LIN {X 0,Y 347.807,Z 587.248,A -85,B 0,C 180,E1 -13735.5,E2 -13735.5} C_VEL
LIN {X 0,Y 350.643,Z 598.741,A -85,B 0,C 180,E1 -13738.593,E2 -13738.593} C_VEL
LIN {X 0,Y 352.837,Z 609.241,A -85,B 0,C 180,E1 -13741.213,E2 -13741.213} C_VEL
LIN {X 0,Y 353.457,Z 613.128,A -85,B 0,C 180,E1 -13742.144,E2 -13742.144} C_VEL
LIN {X 0,Y 351.63,Z 628.965,A -85,B 0,C 180,E1 -13745.498,E2 -13745.498} C_VEL
LIN {X 0,Y 351.249,Z 632.568,A -85,B 0,C 180,E1 -13746.255,E2 -13746.255} C_VEL
LIN {X 0,Y 354.896,Z 654.897,A -85,B 0,C 180,E1 -13747.117,E2 -13747.117} C_VEL
LIN {X 0,Y 357.589,Z 678.434,A -85,B 0,C 180,E1 -13747.895,E2 -13747.895} C_VEL
LIN {X 0,Y 355.994,Z 743.795,A -85,B 0,C 180,E1 -13749.374,E2 -13749.374} C_VEL
LIN {X 0,Y 355.12,Z 757.95,A -85,B 0,C 180,E1 -13749.926,E2 -13749.926} C_VEL
LIN {X 0,Y 353.991,Z 770.595,A -85,B 0,C 180,E1 -13750.652,E2 -13750.652} C_VEL
LIN {X 0,Y 352.711,Z 782.342,A -85,B 0,C 180,E1 -13751.56,E2 -13751.56} C_VEL
LIN {X 0,Y 351.401,Z 793.761,A -85,B 0,C 180,E1 -13752.693,E2 -13752.693} C_VEL
LIN {X 0,Y 350.119,Z 804.328,A -85,B 0,C 180,E1 -13754.008,E2 -13754.008} C_VEL
LIN {X 0,Y 349.136,Z 813.806,A -85,B 0,C 180,E1 -13755.478,E2 -13755.478} C_VEL
LIN {X 0,Y 348.13,Z 821.311,A -85,B 0,C 180,E1 -13756.873,E2 -13756.873} C_VEL
LIN {X 0,Y 347.268,Z 829.004,A -85,B 0,C 180,E1 -13758.62,E2 -13758.62} C_VEL
LIN {X 0,Y 346.713,Z 836.139,A -85,B 0,C 180,E1 -13760.668,E2 -13760.668} C_VEL
LIN {X 0,Y 346.519,Z 840.885,A -85,B 0,C 180,E1 -13762.425,E2 -13762.425} C_VEL
LIN {X 0,Y 346.403,Z 844.523,A -85,B 0,C 180,E1 -13764.178,E2 -13764.178} C_VEL
LIN {X 0,Y 346.411,Z 846.353,A -85,B 0,C 180,E1 -13765.345,E2 -13765.345} C_VEL
LIN {X 0,Y 346.594,Z 848.779,A -85,B 0,C 180,E1 -13767.676,E2 -13767.676} C_VEL
LIN {X 0,Y 346.623,Z 849.329,A -85,B 0,C 180,E1 -13768.838,E2 -13768.838} C_VEL
LIN {X 0,Y 346.681,Z 849.46,A -85,B 0,C 180,E1 -13770,E2 -13770} C_VEL
LIN {X 0,Y 346.667,Z 849.18,A -85,B 0,C 180,E1 -13771.162,E2 -13771.162} C_VEL
LIN {X 0,Y 346.617,Z 848.487,A -85,B 0,C 180,E1 -13772.324,E2 -13772.324} C_VEL
LIN {X 0,Y 346.504,Z 847.324,A -85,B 0,C 180,E1 -13773.488,E2 -13773.488} C_VEL
LIN {X 0,Y 346.468,Z 844.785,A -85,B 0,C 180,E1 -13775.237,E2 -13775.237} C_VEL
LIN {X 0,Y 346.469,Z 840.184,A -85,B 0,C 180,E1 -13777.576,E2 -13777.576} C_VEL
LIN {X 0,Y 346.71,Z 835.733,A -85,B 0,C 180,E1 -13779.332,E2 -13779.332} C_VEL
LIN {X 0,Y 347.166,Z 830.086,A -85,B 0,C 180,E1 -13781.088,E2 -13781.088} C_VEL
LIN {X 0,Y 348.039,Z 823.071,A -85,B 0,C 180,E1 -13782.834,E2 -13782.834} C_VEL
LIN {X 0,Y 349.063,Z 814.841,A -85,B 0,C 180,E1 -13784.478,E2 -13784.478} C_VEL
LIN {X 0,Y 350.151,Z 805.338,A -85,B 0,C 180,E1 -13786.02,E2 -13786.02} C_VEL
LIN {X 0,Y 351.496,Z 795.505,A -85,B 0,C 180,E1 -13787.302,E2 -13787.302} C_VEL
LIN {X 0,Y 352.903,Z 784.628,A -85,B 0,C 180,E1 -13788.43,E2 -13788.43} C_VEL
LIN {X 0,Y 354.156,Z 772.464,A -85,B 0,C 180,E1 -13789.414,E2 -13789.414} C_VEL
LIN {X 0,Y 355.416,Z 759.627,A -85,B 0,C 180,E1 -13790.17,E2 -13790.17} C_VEL
LIN {X 0,Y 356.266,Z 746.66,A -85,B 0,C 180,E1 -13790.685,E2 -13790.685} C_VEL
LIN {X 0,Y 356.74,Z 726.665,A -85,B 0,C 180,E1 -13791.149,E2 -13791.149} C_VEL
LIN {X 0,Y 357.675,Z 675.14,A -85,B 0,C 180,E1 -13792.209,E2 -13792.209} C_VEL
LIN {X 0,Y 354.114,Z 644.038,A -85,B 0,C 180,E1 -13793.174,E2 -13793.174} C_VEL
LIN {X 0,Y 351.817,Z 628.158,A -85,B 0,C 180,E1 -13793.751,E2 -13793.751} C_VEL
LIN {X 0,Y 353.374,Z 612.718,A -85,B 0,C 180,E1 -13796.495,E2 -13796.495} C_VEL
LIN {X 0,Y 352.12,Z 605.557,A -85,B 0,C 180,E1 -13797.901,E2 -13797.901} C_VEL
LIN {X 0,Y 348.167,Z 588.997,A -85,B 0,C 180,E1 -13801.317,E2 -13801.317} C_VEL
LIN {X 0,Y 347.753,Z 587.169,A -85,B 0,C 180,E1 -13801.753,E2 -13801.753} C_VEL
LIN {X 0,Y 347.788,Z 587.165,A -85,B 0,C 180,E1 -13805.874,E2 -13805.874} C_VEL
LIN {X 0,Y 347.764,Z 587.161,A -85,B 0,C 180,E1 -13808.79,E2 -13808.79} C_VEL
LIN {X 0,Y 347.764,Z 587.16,A -85,B 0,C 180,E1 -13811.827,E2 -13811.827} C_VEL
LIN {X 0,Y 347.796,Z 587.157,A -85,B 0,C 180,E1 -13815.011,E2 -13815.011} C_VEL
LIN {X 0,Y 347.78,Z 587.163,A -85,B 0,C 180,E1 -13818.39,E2 -13818.39} C_VEL
LIN {X 0,Y 347.774,Z 587.162,A -85,B 0,C 180,E1 -13822.009,E2 -13822.009} C_VEL
LIN {X 0,Y 347.739,Z 587.154,A -85,B 0,C 180,E1 -13825.535,E2 -13825.535} C_VEL
LIN {X 0,Y 347.758,Z 587.169,A -85,B 0,C 180,E1 -13828.302,E2 -13828.302} C_VEL
LIN {X 0,Y 347.8,Z 587.145,A -85,B 0,C 180,E1 -13830.989,E2 -13830.989} C_VEL
LIN {X 0,Y 347.825,Z 587.156,A -85,B 0,C 180,E1 -13833.607,E2 -13833.607} C_VEL
LIN {X 0,Y 347.781,Z 587.153,A -85,B 0,C 180,E1 -13836.161,E2 -13836.161} C_VEL
LIN {X 0,Y 347.805,Z 587.158,A -85,B 0,C 180,E1 -13839.909,E2 -13839.909} C_VEL
LIN {X 0,Y 347.858,Z 587.147,A -85,B 0,C 180,E1 -13842.359,E2 -13842.359} C_VEL
LIN {X 0,Y 347.89,Z 587.142,A -85,B 0,C 180,E1 -13845.97,E2 -13845.97} C_VEL
LIN {X 0,Y 347.921,Z 587.137,A -85,B 0,C 180,E1 -13849.525,E2 -13849.525} C_VEL
LIN {X 0,Y 348.086,Z 587.121,A -85,B 0,C 180,E1 -13853.042,E2 -13853.042} C_VEL
LIN {X 0,Y 348.201,Z 587.095,A -85,B 0,C 180,E1 -13857.686,E2 -13857.686} C_VEL
LIN {X 0,Y 348.339,Z 587.084,A -85,B 0,C 180,E1 -13860,E2 -13860} C_VEL
LIN {X 0,Y 348.2,Z 587.111,A -85,B 0,C 180,E1 -13862.314,E2 -13862.314} C_VEL
LIN {X 0,Y 348.085,Z 587.114,A -85,B 0,C 180,E1 -13866.958,E2 -13866.958} C_VEL
LIN {X 0,Y 347.92,Z 587.145,A -85,B 0,C 180,E1 -13870.475,E2 -13870.475} C_VEL
LIN {X 0,Y 347.891,Z 587.142,A -85,B 0,C 180,E1 -13874.15,E2 -13874.15} C_VEL
LIN {X 0,Y 347.884,Z 587.14,A -85,B 0,C 180,E1 -13878.291,E2 -13878.291} C_VEL
LIN {X 0,Y 347.778,Z 587.163,A -85,B 0,C 180,E1 -13881.634,E2 -13881.634} C_VEL
LIN {X 0,Y 347.804,Z 587.15,A -85,B 0,C 180,E1 -13885.109,E2 -13885.109} C_VEL
LIN {X 0,Y 347.806,Z 587.159,A -85,B 0,C 180,E1 -13887.694,E2 -13887.694} C_VEL
LIN {X 0,Y 347.765,Z 587.155,A -85,B 0,C 180,E1 -13890.347,E2 -13890.347} C_VEL
LIN {X 0,Y 347.743,Z 587.159,A -85,B 0,C 180,E1 -13894.045,E2 -13894.045} C_VEL
LIN {X 0,Y 347.758,Z 587.166,A -85,B 0,C 180,E1 -13897.321,E2 -13897.321} C_VEL
LIN {X 0,Y 347.751,Z 587.161,A -85,B 0,C 180,E1 -13900.295,E2 -13900.295} C_VEL
LIN {X 0,Y 347.74,Z 587.15,A -85,B 0,C 180,E1 -13903.406,E2 -13903.406} C_VEL
LIN {X 0,Y 347.725,Z 587.16,A -85,B 0,C 180,E1 -13906.687,E2 -13906.687} C_VEL
LIN {X 0,Y 347.745,Z 587.169,A -85,B 0,C 180,E1 -13910.174,E2 -13910.174} C_VEL
LIN {X 0,Y 347.76,Z 587.156,A -85,B 0,C 180,E1 -13912.68,E2 -13912.68} C_VEL
LIN {X 0,Y 347.77,Z 587.166,A -85,B 0,C 180,E1 -13913.935,E2 -13913.935} C_VEL
LIN {X 0,Y 348.878,Z 590.169,A -85,B 0,C 180,E1 -13914.134,E2 -13914.134} C_VEL
LIN {X 0,Y 356.945,Z 606.471,A -85,B 0,C 180,E1 -13915.183,E2 -13915.183} C_VEL
LIN {X 0,Y 359.514,Z 612.214,A -85,B 0,C 180,E1 -13915.517,E2 -13915.517} C_VEL
LIN {X 0,Y 357.936,Z 684.333,A -85,B 0,C 180,E1 -13916.986,E2 -13916.986} C_VEL
LIN {X 0,Y 357.54,Z 697.812,A -85,B 0,C 180,E1 -13917.464,E2 -13917.464} C_VEL
LIN {X 0,Y 356.928,Z 709.71,A -85,B 0,C 180,E1 -13918.099,E2 -13918.099} C_VEL
LIN {X 0,Y 355.97,Z 721.495,A -85,B 0,C 180,E1 -13918.95,E2 -13918.95} C_VEL
LIN {X 0,Y 354.873,Z 732.621,A -85,B 0,C 180,E1 -13919.997,E2 -13919.997} C_VEL
LIN {X 0,Y 353.582,Z 743.445,A -85,B 0,C 180,E1 -13921.279,E2 -13921.279} C_VEL
LIN {X 0,Y 352.312,Z 752.919,A -85,B 0,C 180,E1 -13922.69,E2 -13922.69} C_VEL
LIN {X 0,Y 351.113,Z 761.41,A -85,B 0,C 180,E1 -13924.255,E2 -13924.255} C_VEL
LIN {X 0,Y 349.923,Z 769.073,A -85,B 0,C 180,E1 -13926.002,E2 -13926.002} C_VEL
LIN {X 0,Y 348.877,Z 775.646,A -85,B 0,C 180,E1 -13927.919,E2 -13927.919} C_VEL
LIN {X 0,Y 348.027,Z 780.921,A -85,B 0,C 180,E1 -13929.923,E2 -13929.923} C_VEL
LIN {X 0,Y 347.426,Z 784.785,A -85,B 0,C 180,E1 -13931.944,E2 -13931.944} C_VEL
LIN {X 0,Y 347.024,Z 786.887,A -85,B 0,C 180,E1 -13933.529,E2 -13933.529} C_VEL
LIN {X 0,Y 346.831,Z 787.974,A -85,B 0,C 180,E1 -13934.727,E2 -13934.727} C_VEL
LIN {X 0,Y 346.636,Z 788.884,A -85,B 0,C 180,E1 -13937.114,E2 -13937.114} C_VEL
LIN {X 0,Y 346.584,Z 788.745,A -85,B 0,C 180,E1 -13938.301,E2 -13938.301} C_VEL
LIN {X 0,Y 346.634,Z 787.198,A -85,B 0,C 180,E1 -13940.666,E2 -13940.666} C_VEL
LIN {X 0,Y 346.765,Z 785.836,A -85,B 0,C 180,E1 -13941.844,E2 -13941.844} C_VEL
LIN {X 0,Y 347.064,Z 782.957,A -85,B 0,C 180,E1 -13943.606,E2 -13943.606} C_VEL
LIN {X 0,Y 347.388,Z 779.064,A -85,B 0,C 180,E1 -13945.358,E2 -13945.358} C_VEL
LIN {X 0,Y 347.813,Z 774.039,A -85,B 0,C 180,E1 -13947.105,E2 -13947.105} C_VEL
LIN {X 0,Y 348.499,Z 767.685,A -85,B 0,C 180,E1 -13948.844,E2 -13948.844} C_VEL
LIN {X 0,Y 349.282,Z 759.809,A -85,B 0,C 180,E1 -13950.576,E2 -13950.576} C_VEL
LIN {X 0,Y 350.172,Z 751.746,A -85,B 0,C 180,E1 -13952.013,E2 -13952.013} C_VEL
LIN {X 0,Y 351.115,Z 741.892,A -85,B 0,C 180,E1 -13953.443,E2 -13953.443} C_VEL
LIN {X 0,Y 352.091,Z 730.83,A -85,B 0,C 180,E1 -13954.723,E2 -13954.723} C_VEL
LIN {X 0,Y 352.973,Z 720.002,A -85,B 0,C 180,E1 -13955.713,E2 -13955.713} C_VEL
LIN {X 0,Y 353.669,Z 707.954,A -85,B 0,C 180,E1 -13956.561,E2 -13956.561} C_VEL
LIN {X 0,Y 354.218,Z 694.721,A -85,B 0,C 180,E1 -13957.231,E2 -13957.231} C_VEL
LIN {X 0,Y 354.53,Z 682.914,A -85,B 0,C 180,E1 -13957.618,E2 -13957.618} C_VEL
LIN {X 0,Y 355.717,Z 608.285,A -85,B 0,C 180,E1 -13959.124,E2 -13959.124} C_VEL
LIN {X 0,Y 350.334,Z 593.661,A -85,B 0,C 180,E1 -13959.725,E2 -13959.725} C_VEL
LIN {X 0,Y 347.964,Z 587.144,A -85,B 0,C 180,E1 -13960.005,E2 -13960.005} C_VEL
LIN {X 0,Y 347.9,Z 587.152,A -85,B 0,C 180,E1 -13964.149,E2 -13964.149} C_VEL
LIN {X 0,Y 347.893,Z 587.152,A -85,B 0,C 180,E1 -13968.29,E2 -13968.29} C_VEL
LIN {X 0,Y 347.867,Z 587.153,A -85,B 0,C 180,E1 -13968.634,E2 -13968.634} C_VEL
LIN {X 0,Y 347.161,Z 587.24,A -85,B 0,C 180,E1 -13969.277,E2 -13969.277} C_VEL
LIN {X 0,Y 344.285,Z 587.601,A -85,B 0,C 180,E1 -13970.284,E2 -13970.284} C_VEL
LIN {X 0,Y 341.403,Z 587.961,A -85,B 0,C 180,E1 -13971.307,E2 -13971.307} C_VEL
LIN {X 0,Y 340.714,Z 588.043,A -85,B 0,C 180,E1 -13971.968,E2 -13971.968} C_VEL
LIN {X 0,Y 340.75,Z 588.037,A -85,B 0,C 180,E1 -13973.203,E2 -13973.203} C_VEL
LIN {X 0,Y 342.594,Z 592.979,A -85,B 0,C 180,E1 -13973.467,E2 -13973.467} C_VEL
LIN {X 0,Y 349.529,Z 610.359,A -85,B 0,C 180,E1 -13974.303,E2 -13974.303} C_VEL
LIN {X 0,Y 348.094,Z 679.063,A -85,B 0,C 180,E1 -13975.827,E2 -13975.827} C_VEL
LIN {X 0,Y 347.807,Z 692.389,A -85,B 0,C 180,E1 -13976.232,E2 -13976.232} C_VEL
LIN {X 0,Y 347.322,Z 705.35,A -85,B 0,C 180,E1 -13976.862,E2 -13976.862} C_VEL
LIN {X 0,Y 346.562,Z 717.77,A -85,B 0,C 180,E1 -13977.698,E2 -13977.698} C_VEL
LIN {X 0,Y 345.658,Z 729.584,A -85,B 0,C 180,E1 -13978.757,E2 -13978.757} C_VEL
LIN {X 0,Y 344.684,Z 740.315,A -85,B 0,C 180,E1 -13979.969,E2 -13979.969} C_VEL
LIN {X 0,Y 343.71,Z 749.983,A -85,B 0,C 180,E1 -13981.319,E2 -13981.319} C_VEL
LIN {X 0,Y 342.79,Z 758.591,A -85,B 0,C 180,E1 -13982.797,E2 -13982.797} C_VEL
LIN {X 0,Y 341.802,Z 767.365,A -85,B 0,C 180,E1 -13984.667,E2 -13984.667} C_VEL
LIN {X 0,Y 341.077,Z 774.28,A -85,B 0,C 180,E1 -13986.524,E2 -13986.524} C_VEL
LIN {X 0,Y 340.513,Z 779.599,A -85,B 0,C 180,E1 -13988.344,E2 -13988.344} C_VEL
LIN {X 0,Y 340.045,Z 783.622,A -85,B 0,C 180,E1 -13990.118,E2 -13990.118} C_VEL
LIN {X 0,Y 339.736,Z 786.566,A -85,B 0,C 180,E1 -13991.865,E2 -13991.865} C_VEL
LIN {X 0,Y 339.522,Z 788.538,A -85,B 0,C 180,E1 -13993.573,E2 -13993.573} C_VEL
LIN {X 0,Y 339.434,Z 789.629,A -85,B 0,C 180,E1 -13995.253,E2 -13995.253} C_VEL
LIN {X 0,Y 339.498,Z 789.921,A -85,B 0,C 180,E1 -13996.911,E2 -13996.911} C_VEL
LIN {X 0,Y 339.603,Z 789.475,A -85,B 0,C 180,E1 -13998.53,E2 -13998.53} C_VEL
LIN {X 0,Y 339.869,Z 788.279,A -85,B 0,C 180,E1 -14000.131,E2 -14000.131} C_VEL
LIN {X 0,Y 340.447,Z 785.112,A -85,B 0,C 180,E1 -14002.484,E2 -14002.484} C_VEL
LIN {X 0,Y 340.931,Z 781.817,A -85,B 0,C 180,E1 -14004.156,E2 -14004.156} C_VEL
LIN {X 0,Y 341.775,Z 776.211,A -85,B 0,C 180,E1 -14006.275,E2 -14006.275} C_VEL
LIN {X 0,Y 342.784,Z 769.782,A -85,B 0,C 180,E1 -14008.133,E2 -14008.133} C_VEL
LIN {X 0,Y 343.98,Z 761.685,A -85,B 0,C 180,E1 -14009.966,E2 -14009.966} C_VEL
LIN {X 0,Y 345.111,Z 753.319,A -85,B 0,C 180,E1 -14011.494,E2 -14011.494} C_VEL
LIN {X 0,Y 346.508,Z 742.896,A -85,B 0,C 180,E1 -14013.019,E2 -14013.019} C_VEL
LIN {X 0,Y 347.632,Z 732.479,A -85,B 0,C 180,E1 -14014.236,E2 -14014.236} C_VEL
LIN {X 0,Y 348.706,Z 721.132,A -85,B 0,C 180,E1 -14015.29,E2 -14015.29} C_VEL
LIN {X 0,Y 349.631,Z 709.216,A -85,B 0,C 180,E1 -14016.138,E2 -14016.138} C_VEL
LIN {X 0,Y 350.174,Z 696.584,A -85,B 0,C 180,E1 -14016.797,E2 -14016.797} C_VEL
LIN {X 0,Y 350.531,Z 684.532,A -85,B 0,C 180,E1 -14017.209,E2 -14017.209} C_VEL
LIN {X 0,Y 352.43,Z 613.13,A -85,B 0,C 180,E1 -14018.855,E2 -14018.855} C_VEL
LIN {X 0,Y 345.875,Z 598.906,A -85,B 0,C 180,E1 -14019.792,E2 -14019.792} C_VEL
LIN {X 0,Y 340.992,Z 589.133,A -85,B 0,C 180,E1 -14020.511,E2 -14020.511} C_VEL
LIN {X 0,Y 340.769,Z 588.039,A -85,B 0,C 180,E1 -14020.576,E2 -14020.576} C_VEL
LIN {X 0,Y 340.779,Z 588.036,A -85,B 0,C 180,E1 -14023.218,E2 -14023.218} C_VEL
LIN {X 0,Y 340.839,Z 588.03,A -85,B 0,C 180,E1 -14026.89,E2 -14026.89} C_VEL
LIN {X 0,Y 340.922,Z 588.017,A -85,B 0,C 180,E1 -14030.508,E2 -14030.508} C_VEL
LIN {X 0,Y 341.07,Z 587.999,A -85,B 0,C 180,E1 -14032.898,E2 -14032.898} C_VEL
LIN {X 0,Y 341.163,Z 587.983,A -85,B 0,C 180,E1 -14037.639,E2 -14037.639} C_VEL
LIN {X 0,Y 341.309,Z 587.969,A -85,B 0,C 180,E1 -14040,E2 -14040} C_VEL
LIN {X 0,Y 341.162,Z 587.99,A -85,B 0,C 180,E1 -14042.361,E2 -14042.361} C_VEL
LIN {X 0,Y 341.057,Z 587.994,A -85,B 0,C 180,E1 -14047.102,E2 -14047.102} C_VEL
LIN {X 0,Y 340.867,Z 588.017,A -85,B 0,C 180,E1 -14050.694,E2 -14050.694} C_VEL
LIN {X 0,Y 340.856,Z 588.016,A -85,B 0,C 180,E1 -14054.325,E2 -14054.325} C_VEL
LIN {X 0,Y 340.831,Z 588.025,A -85,B 0,C 180,E1 -14058.467,E2 -14058.467} C_VEL
LIN {X 0,Y 340.747,Z 588.036,A -85,B 0,C 180,E1 -14061.857,E2 -14061.857} C_VEL
LIN {X 0,Y 340.766,Z 588.036,A -85,B 0,C 180,E1 -14065.665,E2 -14065.665} C_VEL
LIN {X 0,Y 340.736,Z 588.038,A -85,B 0,C 180,E1 -14068.32,E2 -14068.32} C_VEL
LIN {X 0,Y 340.699,Z 588.043,A -85,B 0,C 180,E1 -14071.045,E2 -14071.045} C_VEL
LIN {X 0,Y 340.713,Z 588.044,A -85,B 0,C 180,E1 -14075.28,E2 -14075.28} C_VEL
LIN {X 0,Y 340.714,Z 588.045,A -85,B 0,C 180,E1 -14078.389,E2 -14078.389} C_VEL
LIN {X 0,Y 340.721,Z 588.04,A -85,B 0,C 180,E1 -14081.305,E2 -14081.305} C_VEL
LIN {X 0,Y 340.718,Z 588.045,A -85,B 0,C 180,E1 -14084.533,E2 -14084.533} C_VEL
LIN {X 0,Y 340.731,Z 588.043,A -85,B 0,C 180,E1 -14087.949,E2 -14087.949} C_VEL
LIN {X 0,Y 340.737,Z 588.043,A -85,B 0,C 180,E1 -14091.774,E2 -14091.774} C_VEL
LIN {X 0,Y 340.75,Z 588.112,A -85,B 0,C 180,E1 -14094.905,E2 -14094.905} C_VEL
LIN {X 0,Y 343.72,Z 599.975,A -85,B 0,C 180,E1 -14098.208,E2 -14098.208} C_VEL
LIN {X 0,Y 345.889,Z 610.372,A -85,B 0,C 180,E1 -14100.892,E2 -14100.892} C_VEL
LIN {X 0,Y 346.584,Z 614.357,A -85,B 0,C 180,E1 -14101.872,E2 -14101.872} C_VEL
LIN {X 0,Y 345.433,Z 624.369,A -85,B 0,C 180,E1 -14104.061,E2 -14104.061} C_VEL
LIN {X 0,Y 344.559,Z 631.889,A -85,B 0,C 180,E1 -14105.675,E2 -14105.675} C_VEL
LIN {X 0,Y 348.333,Z 654.595,A -85,B 0,C 180,E1 -14106.582,E2 -14106.582} C_VEL
LIN {X 0,Y 351.166,Z 679.683,A -85,B 0,C 180,E1 -14107.442,E2 -14107.442} C_VEL
LIN {X 0,Y 349.433,Z 743.746,A -85,B 0,C 180,E1 -14108.93,E2 -14108.93} C_VEL
LIN {X 0,Y 348.535,Z 757.689,A -85,B 0,C 180,E1 -14109.491,E2 -14109.491} C_VEL
LIN {X 0,Y 347.438,Z 769.695,A -85,B 0,C 180,E1 -14110.196,E2 -14110.196} C_VEL
LIN {X 0,Y 345.997,Z 782.284,A -85,B 0,C 180,E1 -14111.189,E2 -14111.189} C_VEL
LIN {X 0,Y 344.639,Z 793.599,A -85,B 0,C 180,E1 -14112.342,E2 -14112.342} C_VEL
LIN {X 0,Y 343.274,Z 803.848,A -85,B 0,C 180,E1 -14113.65,E2 -14113.65} C_VEL
LIN {X 0,Y 342.186,Z 813.814,A -85,B 0,C 180,E1 -14115.241,E2 -14115.241} C_VEL
LIN {X 0,Y 341.008,Z 822.306,A -85,B 0,C 180,E1 -14116.897,E2 -14116.897} C_VEL
LIN {X 0,Y 340.158,Z 829.688,A -85,B 0,C 180,E1 -14118.681,E2 -14118.681} C_VEL
LIN {X 0,Y 339.675,Z 835.625,A -85,B 0,C 180,E1 -14120.473,E2 -14120.473} C_VEL
LIN {X 0,Y 339.429,Z 840.345,A -85,B 0,C 180,E1 -14122.266,E2 -14122.266} C_VEL
LIN {X 0,Y 339.327,Z 843.962,A -85,B 0,C 180,E1 -14124.056,E2 -14124.056} C_VEL
LIN {X 0,Y 339.341,Z 845.783,A -85,B 0,C 180,E1 -14125.248,E2 -14125.248} C_VEL
LIN {X 0,Y 339.525,Z 848.183,A -85,B 0,C 180,E1 -14127.627,E2 -14127.627} C_VEL
LIN {X 0,Y 339.551,Z 848.71,A -85,B 0,C 180,E1 -14128.814,E2 -14128.814} C_VEL
LIN {X 0,Y 339.636,Z 848.831,A -85,B 0,C 180,E1 -14130,E2 -14130} C_VEL
LIN {X 0,Y 339.593,Z 848.535,A -85,B 0,C 180,E1 -14131.186,E2 -14131.186} C_VEL
LIN {X 0,Y 339.55,Z 847.823,A -85,B 0,C 180,E1 -14132.372,E2 -14132.372} C_VEL
LIN {X 0,Y 339.416,Z 846.631,A -85,B 0,C 180,E1 -14133.561,E2 -14133.561} C_VEL
LIN {X 0,Y 339.377,Z 842.529,A -85,B 0,C 180,E1 -14136.272,E2 -14136.272} C_VEL
LIN {X 0,Y 339.467,Z 838.381,A -85,B 0,C 180,E1 -14138.333,E2 -14138.333} C_VEL
LIN {X 0,Y 339.8,Z 833.591,A -85,B 0,C 180,E1 -14140.125,E2 -14140.125} C_VEL
LIN {X 0,Y 340.452,Z 827.551,A -85,B 0,C 180,E1 -14141.913,E2 -14141.913} C_VEL
LIN {X 0,Y 341.349,Z 820.058,A -85,B 0,C 180,E1 -14143.696,E2 -14143.696} C_VEL
LIN {X 0,Y 342.453,Z 811.741,A -85,B 0,C 180,E1 -14145.299,E2 -14145.299} C_VEL
LIN {X 0,Y 343.792,Z 802.168,A -85,B 0,C 180,E1 -14146.783,E2 -14146.783} C_VEL
LIN {X 0,Y 345.235,Z 791.706,A -85,B 0,C 180,E1 -14148.086,E2 -14148.086} C_VEL
LIN {X 0,Y 346.7,Z 780.07,A -85,B 0,C 180,E1 -14149.232,E2 -14149.232} C_VEL
LIN {X 0,Y 347.989,Z 768.75,A -85,B 0,C 180,E1 -14150.079,E2 -14150.079} C_VEL
LIN {X 0,Y 349.125,Z 756.052,A -85,B 0,C 180,E1 -14150.78,E2 -14150.78} C_VEL
LIN {X 0,Y 349.929,Z 743.308,A -85,B 0,C 180,E1 -14151.251,E2 -14151.251} C_VEL
LIN {X 0,Y 351.265,Z 675.932,A -85,B 0,C 180,E1 -14152.686,E2 -14152.686} C_VEL
LIN {X 0,Y 348.077,Z 647.6,A -85,B 0,C 180,E1 -14153.584,E2 -14153.584} C_VEL
LIN {X 0,Y 345.076,Z 626.818,A -85,B 0,C 180,E1 -14154.324,E2 -14154.324} C_VEL
LIN {X 0,Y 346.423,Z 613.264,A -85,B 0,C 180,E1 -14156.792,E2 -14156.792} C_VEL
LIN {X 0,Y 343.939,Z 601.661,A -85,B 0,C 180,E1 -14159.156,E2 -14159.156} C_VEL
LIN {X 0,Y 340.702,Z 588.048,A -85,B 0,C 180,E1 -14162.084,E2 -14162.084} C_VEL
LIN {X 0,Y 340.717,Z 588.043,A -85,B 0,C 180,E1 -14165.278,E2 -14165.278} C_VEL
LIN {X 0,Y 340.717,Z 588.038,A -85,B 0,C 180,E1 -14168.387,E2 -14168.387} C_VEL
LIN {X 0,Y 340.73,Z 588.036,A -85,B 0,C 180,E1 -14172.051,E2 -14172.051} C_VEL
LIN {X 0,Y 340.719,Z 588.036,A -85,B 0,C 180,E1 -14175.467,E2 -14175.467} C_VEL
LIN {X 0,Y 340.721,Z 588.04,A -85,B 0,C 180,E1 -14178.695,E2 -14178.695} C_VEL
LIN {X 0,Y 340.736,Z 588.036,A -85,B 0,C 180,E1 -14181.773,E2 -14181.773} C_VEL
LIN {X 0,Y 340.718,Z 588.028,A -85,B 0,C 180,E1 -14185.595,E2 -14185.595} C_VEL
LIN {X 0,Y 340.71,Z 588.041,A -85,B 0,C 180,E1 -14188.956,E2 -14188.956} C_VEL
LIN {X 0,Y 340.773,Z 588.029,A -85,B 0,C 180,E1 -14192.473,E2 -14192.473} C_VEL
LIN {X 0,Y 340.749,Z 588.035,A -85,B 0,C 180,E1 -14195.638,E2 -14195.638} C_VEL
LIN {X 0,Y 340.738,Z 588.037,A -85,B 0,C 180,E1 -14199.474,E2 -14199.474} C_VEL
LIN {X 0,Y 340.85,Z 588.026,A -85,B 0,C 180,E1 -14201.984,E2 -14201.984} C_VEL
LIN {X 0,Y 340.862,Z 588.017,A -85,B 0,C 180,E1 -14205.705,E2 -14205.705} C_VEL
LIN {X 0,Y 340.863,Z 588.017,A -85,B 0,C 180,E1 -14209.306,E2 -14209.306} C_VEL
LIN {X 0,Y 341.054,Z 587.994,A -85,B 0,C 180,E1 -14212.898,E2 -14212.898} C_VEL
LIN {X 0,Y 341.163,Z 587.972,A -85,B 0,C 180,E1 -14217.639,E2 -14217.639} C_VEL
LIN {X 0,Y 341.289,Z 587.962,A -85,B 0,C 180,E1 -14220,E2 -14220} C_VEL
LIN {X 0,Y 341.162,Z 587.989,A -85,B 0,C 180,E1 -14222.361,E2 -14222.361} C_VEL
LIN {X 0,Y 341.053,Z 587.991,A -85,B 0,C 180,E1 -14227.102,E2 -14227.102} C_VEL
LIN {X 0,Y 340.863,Z 588.02,A -85,B 0,C 180,E1 -14230.694,E2 -14230.694} C_VEL
LIN {X 0,Y 340.856,Z 588.019,A -85,B 0,C 180,E1 -14234.325,E2 -14234.325} C_VEL
LIN {X 0,Y 340.83,Z 588.016,A -85,B 0,C 180,E1 -14238.467,E2 -14238.467} C_VEL
LIN {X 0,Y 340.747,Z 588.038,A -85,B 0,C 180,E1 -14241.857,E2 -14241.857} C_VEL
LIN {X 0,Y 340.765,Z 588.031,A -85,B 0,C 180,E1 -14245.665,E2 -14245.665} C_VEL
LIN {X 0,Y 340.736,Z 588.039,A -85,B 0,C 180,E1 -14248.32,E2 -14248.32} C_VEL
LIN {X 0,Y 340.71,Z 588.039,A -85,B 0,C 180,E1 -14251.044,E2 -14251.044} C_VEL
LIN {X 0,Y 340.713,Z 588.039,A -85,B 0,C 180,E1 -14255.28,E2 -14255.28} C_VEL
LIN {X 0,Y 340.713,Z 588.043,A -85,B 0,C 180,E1 -14258.388,E2 -14258.388} C_VEL
LIN {X 0,Y 340.727,Z 588.013,A -85,B 0,C 180,E1 -14262.052,E2 -14262.052} C_VEL
LIN {X 0,Y 340.681,Z 588.049,A -85,B 0,C 180,E1 -14265.462,E2 -14265.462} C_VEL
LIN {X 0,Y 340.683,Z 588.035,A -85,B 0,C 180,E1 -14268.691,E2 -14268.691} C_VEL
LIN {X 0,Y 340.731,Z 588.029,A -85,B 0,C 180,E1 -14271.774,E2 -14271.774} C_VEL
LIN {X 0,Y 340.708,Z 588.042,A -85,B 0,C 180,E1 -14273.339,E2 -14273.339} C_VEL
LIN {X 0,Y 341.743,Z 590.947,A -85,B 0,C 180,E1 -14273.511,E2 -14273.511} C_VEL
LIN {X 0,Y 349.198,Z 605.498,A -85,B 0,C 180,E1 -14274.513,E2 -14274.513} C_VEL
LIN {X 0,Y 353.083,Z 613.998,A -85,B 0,C 180,E1 -14275.033,E2 -14275.033} C_VEL
LIN {X 0,Y 351.511,Z 685.25,A -85,B 0,C 180,E1 -14276.517,E2 -14276.517} C_VEL
LIN {X 0,Y 351.122,Z 698.274,A -85,B 0,C 180,E1 -14276.989,E2 -14276.989} C_VEL
LIN {X 0,Y 350.404,Z 711.311,A -85,B 0,C 180,E1 -14277.706,E2 -14277.706} C_VEL
LIN {X 0,Y 349.335,Z 723.519,A -85,B 0,C 180,E1 -14278.631,E2 -14278.631} C_VEL
LIN {X 0,Y 348.059,Z 735.458,A -85,B 0,C 180,E1 -14279.814,E2 -14279.814} C_VEL
LIN {X 0,Y 346.608,Z 746.437,A -85,B 0,C 180,E1 -14281.213,E2 -14281.213} C_VEL
LIN {X 0,Y 345.285,Z 756.017,A -85,B 0,C 180,E1 -14282.745,E2 -14282.745} C_VEL
LIN {X 0,Y 343.844,Z 765.113,A -85,B 0,C 180,E1 -14284.582,E2 -14284.582} C_VEL
LIN {X 0,Y 342.653,Z 772.362,A -85,B 0,C 180,E1 -14286.425,E2 -14286.425} C_VEL
LIN {X 0,Y 341.704,Z 778.054,A -85,B 0,C 180,E1 -14288.272,E2 -14288.272} C_VEL
LIN {X 0,Y 340.919,Z 782.444,A -85,B 0,C 180,E1 -14290.115,E2 -14290.115} C_VEL
LIN {X 0,Y 340.364,Z 785.694,A -85,B 0,C 180,E1 -14291.958,E2 -14291.958} C_VEL
LIN {X 0,Y 340.044,Z 787.281,A -85,B 0,C 180,E1 -14293.181,E2 -14293.181} C_VEL
LIN {X 0,Y 339.806,Z 788.455,A -85,B 0,C 180,E1 -14294.403,E2 -14294.403} C_VEL
LIN {X 0,Y 339.586,Z 789.445,A -85,B 0,C 180,E1 -14296.583,E2 -14296.583} C_VEL
LIN {X 0,Y 339.522,Z 789.391,A -85,B 0,C 180,E1 -14298.054,E2 -14298.054} C_VEL
LIN {X 0,Y 339.495,Z 788.893,A -85,B 0,C 180,E1 -14299.263,E2 -14299.263} C_VEL
LIN {X 0,Y 339.681,Z 786.656,A -85,B 0,C 180,E1 -14301.673,E2 -14301.673} C_VEL
LIN {X 0,Y 339.865,Z 784.672,A -85,B 0,C 180,E1 -14303.019,E2 -14303.019} C_VEL
LIN {X 0,Y 340.307,Z 780.084,A -85,B 0,C 180,E1 -14305.262,E2 -14305.262} C_VEL
LIN {X 0,Y 340.728,Z 775.188,A -85,B 0,C 180,E1 -14307.044,E2 -14307.044} C_VEL
LIN {X 0,Y 341.42,Z 768.998,A -85,B 0,C 180,E1 -14308.821,E2 -14308.821} C_VEL
LIN {X 0,Y 342.207,Z 761.267,A -85,B 0,C 180,E1 -14310.588,E2 -14310.588} C_VEL
LIN {X 0,Y 343.326,Z 751.629,A -85,B 0,C 180,E1 -14312.346,E2 -14312.346} C_VEL
LIN {X 0,Y 344.274,Z 741.581,A -85,B 0,C 180,E1 -14313.804,E2 -14313.804} C_VEL
LIN {X 0,Y 345.311,Z 730.322,A -85,B 0,C 180,E1 -14315.108,E2 -14315.108} C_VEL
LIN {X 0,Y 346.243,Z 719.127,A -85,B 0,C 180,E1 -14316.117,E2 -14316.117} C_VEL
LIN {X 0,Y 346.945,Z 706.597,A -85,B 0,C 180,E1 -14316.981,E2 -14316.981} C_VEL
LIN {X 0,Y 347.467,Z 694.264,A -85,B 0,C 180,E1 -14317.591,E2 -14317.591} C_VEL
LIN {X 0,Y 347.779,Z 682.133,A -85,B 0,C 180,E1 -14317.972,E2 -14317.972} C_VEL
LIN {X 0,Y 348.895,Z 609.148,A -85,B 0,C 180,E1 -14319.474,E2 -14319.474} C_VEL
LIN {X 0,Y 341,Z 588.596,A -85,B 0,C 180,E1 -14320.367,E2 -14320.367} C_VEL
LIN {X 0,Y 340.901,Z 588.021,A -85,B 0,C 180,E1 -14320.422,E2 -14320.422} C_VEL
LIN {X 0,Y 340.864,Z 588.027,A -85,B 0,C 180,E1 -14324.324,E2 -14324.324} C_VEL
LIN {X 0,Y 340.825,Z 588.03,A -85,B 0,C 180,E1 -14328.618,E2 -14328.618} C_VEL
LIN {X 0,Y 340.714,Z 588.043,A -85,B 0,C 180,E1 -14331.968,E2 -14331.968} C_VEL
LIN {X 0,Y 340.817,Z 588.682,A -85,B 0,C 180,E1 -14332.405,E2 -14332.405} C_VEL
LIN {X 0,Y 341.178,Z 590.863,A -85,B 0,C 180,E1 -14332.893,E2 -14332.893} C_VEL
LIN {X 0,Y 341.778,Z 594.839,A -85,B 0,C 180,E1 -14333.345,E2 -14333.345} C_VEL
LIN {X 0,Y 342.362,Z 599.598,A -85,B 0,C 180,E1 -14333.614,E2 -14333.614} C_VEL
LIN {X 0,Y 343.211,Z 609.814,A -85,B 0,C 180,E1 -14333.908,E2 -14333.908} C_VEL
LIN {X 0,Y 342.867,Z 616.697,A -85,B 0,C 180,E1 -14334.06,E2 -14334.06} C_VEL
LIN {X 0,Y 341.263,Z 685.918,A -85,B 0,C 180,E1 -14335.645,E2 -14335.645} C_VEL
LIN {X 0,Y 340.819,Z 698.833,A -85,B 0,C 180,E1 -14336.152,E2 -14336.152} C_VEL
LIN {X 0,Y 340.225,Z 711.131,A -85,B 0,C 180,E1 -14336.863,E2 -14336.863} C_VEL
LIN {X 0,Y 339.352,Z 723.36,A -85,B 0,C 180,E1 -14337.809,E2 -14337.809} C_VEL
LIN {X 0,Y 338.354,Z 735.477,A -85,B 0,C 180,E1 -14339.046,E2 -14339.046} C_VEL
LIN {X 0,Y 337.327,Z 745.665,A -85,B 0,C 180,E1 -14340.346,E2 -14340.346} C_VEL
LIN {X 0,Y 336.292,Z 755.189,A -85,B 0,C 180,E1 -14341.848,E2 -14341.848} C_VEL
LIN {X 0,Y 335.395,Z 763.086,A -85,B 0,C 180,E1 -14343.378,E2 -14343.378} C_VEL
LIN {X 0,Y 334.571,Z 769.943,A -85,B 0,C 180,E1 -14344.992,E2 -14344.992} C_VEL
LIN {X 0,Y 333.898,Z 776.414,A -85,B 0,C 180,E1 -14346.885,E2 -14346.885} C_VEL
LIN {X 0,Y 333.321,Z 781.375,A -85,B 0,C 180,E1 -14348.727,E2 -14348.727} C_VEL
LIN {X 0,Y 332.845,Z 785.73,A -85,B 0,C 180,E1 -14350.885,E2 -14350.885} C_VEL
LIN {X 0,Y 332.567,Z 788.083,A -85,B 0,C 180,E1 -14352.549,E2 -14352.549} C_VEL
LIN {X 0,Y 332.396,Z 789.662,A -85,B 0,C 180,E1 -14354.244,E2 -14354.244} C_VEL
LIN {X 0,Y 332.386,Z 790.462,A -85,B 0,C 180,E1 -14355.962,E2 -14355.962} C_VEL
LIN {X 0,Y 332.475,Z 790.456,A -85,B 0,C 180,E1 -14357.717,E2 -14357.717} C_VEL
LIN {X 0,Y 332.696,Z 789.584,A -85,B 0,C 180,E1 -14359.505,E2 -14359.505} C_VEL
LIN {X 0,Y 333.082,Z 787.77,A -85,B 0,C 180,E1 -14361.323,E2 -14361.323} C_VEL
LIN {X 0,Y 333.611,Z 784.916,A -85,B 0,C 180,E1 -14363.178,E2 -14363.178} C_VEL
LIN {X 0,Y 334.339,Z 779.998,A -85,B 0,C 180,E1 -14365.42,E2 -14365.42} C_VEL
LIN {X 0,Y 335.322,Z 774.201,A -85,B 0,C 180,E1 -14367.387,E2 -14367.387} C_VEL
LIN {X 0,Y 336.464,Z 767.317,A -85,B 0,C 180,E1 -14369.216,E2 -14369.216} C_VEL
LIN {X 0,Y 337.778,Z 758.515,A -85,B 0,C 180,E1 -14371.063,E2 -14371.063} C_VEL
LIN {X 0,Y 339.022,Z 749.834,A -85,B 0,C 180,E1 -14372.532,E2 -14372.532} C_VEL
LIN {X 0,Y 340.412,Z 739.223,A -85,B 0,C 180,E1 -14373.978,E2 -14373.978} C_VEL
LIN {X 0,Y 341.681,Z 727.549,A -85,B 0,C 180,E1 -14375.229,E2 -14375.229} C_VEL
LIN {X 0,Y 342.732,Z 715.518,A -85,B 0,C 180,E1 -14376.23,E2 -14376.23} C_VEL
LIN {X 0,Y 343.502,Z 702.549,A -85,B 0,C 180,E1 -14377.024,E2 -14377.024} C_VEL
LIN {X 0,Y 343.986,Z 689.266,A -85,B 0,C 180,E1 -14377.583,E2 -14377.583} C_VEL
LIN {X 0,Y 346.117,Z 615.15,A -85,B 0,C 180,E1 -14379.341,E2 -14379.341} C_VEL
LIN {X 0,Y 339.177,Z 600.225,A -85,B 0,C 180,E1 -14380.382,E2 -14380.382} C_VEL
LIN {X 0,Y 334.08,Z 590.245,A -85,B 0,C 180,E1 -14381.161,E2 -14381.161} C_VEL
LIN {X 0,Y 333.767,Z 588.912,A -85,B 0,C 180,E1 -14381.283,E2 -14381.283} C_VEL
LIN {X 0,Y 333.801,Z 588.907,A -85,B 0,C 180,E1 -14385.576,E2 -14385.576} C_VEL
LIN {X 0,Y 333.83,Z 588.903,A -85,B 0,C 180,E1 -14389.078,E2 -14389.078} C_VEL
LIN {X 0,Y 334.019,Z 588.877,A -85,B 0,C 180,E1 -14392.747,E2 -14392.747} C_VEL
LIN {X 0,Y 333.808,Z 588.902,A -85,B 0,C 180,E1 -14395.169,E2 -14395.169} C_VEL
LIN {X 0,Y 334.1,Z 588.863,A -85,B 0,C 180,E1 -14397.589,E2 -14397.589} C_VEL
LIN {X 0,Y 334.259,Z 588.847,A -85,B 0,C 180,E1 -14400,E2 -14400} C_VEL
LIN {X 0,Y 334.1,Z 588.869,A -85,B 0,C 180,E1 -14402.411,E2 -14402.411} C_VEL
LIN {X 0,Y 334.013,Z 588.877,A -85,B 0,C 180,E1 -14406.039,E2 -14406.039} C_VEL
LIN {X 0,Y 333.977,Z 588.883,A -85,B 0,C 180,E1 -14408.501,E2 -14408.501} C_VEL
LIN {X 0,Y 333.788,Z 588.903,A -85,B 0,C 180,E1 -14412.155,E2 -14412.155} C_VEL
LIN {X 0,Y 333.77,Z 588.903,A -85,B 0,C 180,E1 -14415.887,E2 -14415.887} C_VEL
LIN {X 0,Y 333.79,Z 588.904,A -85,B 0,C 180,E1 -14418.656,E2 -14418.656} C_VEL
LIN {X 0,Y 333.686,Z 588.918,A -85,B 0,C 180,E1 -14422.279,E2 -14422.279} C_VEL
LIN {X 0,Y 333.73,Z 588.915,A -85,B 0,C 180,E1 -14426.247,E2 -14426.247} C_VEL
LIN {X 0,Y 333.706,Z 588.918,A -85,B 0,C 180,E1 -14428.973,E2 -14428.973} C_VEL
LIN {X 0,Y 333.641,Z 588.925,A -85,B 0,C 180,E1 -14432.588,E2 -14432.588} C_VEL
LIN {X 0,Y 333.672,Z 588.92,A -85,B 0,C 180,E1 -14436.14,E2 -14436.14} C_VEL
LIN {X 0,Y 333.68,Z 588.916,A -85,B 0,C 180,E1 -14439.188,E2 -14439.188} C_VEL
LIN {X 0,Y 333.685,Z 588.921,A -85,B 0,C 180,E1 -14442.511,E2 -14442.511} C_VEL
LIN {X 0,Y 333.656,Z 588.924,A -85,B 0,C 180,E1 -14445.966,E2 -14445.966} C_VEL
LIN {X 0,Y 333.654,Z 588.923,A -85,B 0,C 180,E1 -14449.314,E2 -14449.314} C_VEL
LIN {X 0,Y 333.654,Z 588.924,A -85,B 0,C 180,E1 -14452.35,E2 -14452.35} C_VEL
LIN {X 0,Y 333.697,Z 589.062,A -85,B 0,C 180,E1 -14454.3,E2 -14454.3} C_VEL
LIN {X 0,Y 336.51,Z 599.941,A -85,B 0,C 180,E1 -14457.468,E2 -14457.468} C_VEL
LIN {X 0,Y 338.982,Z 611.478,A -85,B 0,C 180,E1 -14460.549,E2 -14460.549} C_VEL
LIN {X 0,Y 339.73,Z 617.018,A -85,B 0,C 180,E1 -14461.926,E2 -14461.926} C_VEL
LIN {X 0,Y 337.874,Z 631.12,A -85,B 0,C 180,E1 -14465.048,E2 -14465.048} C_VEL
LIN {X 0,Y 341.799,Z 654.152,A -85,B 0,C 180,E1 -14466.023,E2 -14466.023} C_VEL
LIN {X 0,Y 344.724,Z 679.551,A -85,B 0,C 180,E1 -14466.924,E2 -14466.924} C_VEL
LIN {X 0,Y 342.964,Z 742.944,A -85,B 0,C 180,E1 -14468.434,E2 -14468.434} C_VEL
LIN {X 0,Y 342.019,Z 756.857,A -85,B 0,C 180,E1 -14469.004,E2 -14469.004} C_VEL
LIN {X 0,Y 340.884,Z 768.871,A -85,B 0,C 180,E1 -14469.72,E2 -14469.72} C_VEL
LIN {X 0,Y 339.462,Z 780.661,A -85,B 0,C 180,E1 -14470.656,E2 -14470.656} C_VEL
LIN {X 0,Y 338.031,Z 792.128,A -85,B 0,C 180,E1 -14471.829,E2 -14471.829} C_VEL
LIN {X 0,Y 336.584,Z 802.562,A -85,B 0,C 180,E1 -14473.16,E2 -14473.16} C_VEL
LIN {X 0,Y 335.408,Z 812.318,A -85,B 0,C 180,E1 -14474.72,E2 -14474.72} C_VEL
LIN {X 0,Y 334.184,Z 820.517,A -85,B 0,C 180,E1 -14476.315,E2 -14476.315} C_VEL
LIN {X 0,Y 333.288,Z 828.122,A -85,B 0,C 180,E1 -14478.136,E2 -14478.136} C_VEL
LIN {X 0,Y 332.749,Z 833.303,A -85,B 0,C 180,E1 -14479.658,E2 -14479.658} C_VEL
LIN {X 0,Y 332.416,Z 838.38,A -85,B 0,C 180,E1 -14481.489,E2 -14481.489} C_VEL
LIN {X 0,Y 332.266,Z 842.32,A -85,B 0,C 180,E1 -14483.32,E2 -14483.32} C_VEL
LIN {X 0,Y 332.273,Z 845.215,A -85,B 0,C 180,E1 -14485.147,E2 -14485.147} C_VEL
LIN {X 0,Y 332.269,Z 846.605,A -85,B 0,C 180,E1 -14486.362,E2 -14486.362} C_VEL
LIN {X 0,Y 332.457,Z 847.583,A -85,B 0,C 180,E1 -14487.577,E2 -14487.577} C_VEL
LIN {X 0,Y 332.482,Z 848.092,A -85,B 0,C 180,E1 -14488.789,E2 -14488.789} C_VEL
LIN {X 0,Y 332.574,Z 848.202,A -85,B 0,C 180,E1 -14490,E2 -14490} C_VEL
LIN {X 0,Y 332.521,Z 847.891,A -85,B 0,C 180,E1 -14491.211,E2 -14491.211} C_VEL
LIN {X 0,Y 332.483,Z 847.153,A -85,B 0,C 180,E1 -14492.423,E2 -14492.423} C_VEL
LIN {X 0,Y 332.303,Z 844.329,A -85,B 0,C 180,E1 -14494.853,E2 -14494.853} C_VEL
LIN {X 0,Y 332.27,Z 840.467,A -85,B 0,C 180,E1 -14497.291,E2 -14497.291} C_VEL
LIN {X 0,Y 332.51,Z 836.48,A -85,B 0,C 180,E1 -14499.121,E2 -14499.121} C_VEL
LIN {X 0,Y 333.038,Z 830.365,A -85,B 0,C 180,E1 -14501.256,E2 -14501.256} C_VEL
LIN {X 0,Y 333.953,Z 823.69,A -85,B 0,C 180,E1 -14503.075,E2 -14503.075} C_VEL
LIN {X 0,Y 335.14,Z 815.351,A -85,B 0,C 180,E1 -14504.903,E2 -14504.903} C_VEL
LIN {X 0,Y 336.181,Z 807.004,A -85,B 0,C 180,E1 -14506.392,E2 -14506.392} C_VEL
LIN {X 0,Y 337.77,Z 796.607,A -85,B 0,C 180,E1 -14507.872,E2 -14507.872} C_VEL
LIN {X 0,Y 339.473,Z 784.925,A -85,B 0,C 180,E1 -14509.187,E2 -14509.187} C_VEL
LIN {X 0,Y 340.855,Z 773.221,A -85,B 0,C 180,E1 -14510.203,E2 -14510.203} C_VEL
LIN {X 0,Y 342.189,Z 761.08,A -85,B 0,C 180,E1 -14510.985,E2 -14510.985} C_VEL
LIN {X 0,Y 343.173,Z 748.719,A -85,B 0,C 180,E1 -14511.552,E2 -14511.552} C_VEL
LIN {X 0,Y 343.687,Z 735.08,A -85,B 0,C 180,E1 -14511.938,E2 -14511.938} C_VEL
LIN {X 0,Y 344.863,Z 676.446,A -85,B 0,C 180,E1 -14513.189,E2 -14513.189} C_VEL
LIN {X 0,Y 341.69,Z 648.033,A -85,B 0,C 180,E1 -14514.117,E2 -14514.117} C_VEL
LIN {X 0,Y 338.409,Z 625.201,A -85,B 0,C 180,E1 -14514.969,E2 -14514.969} C_VEL
LIN {X 0,Y 339.49,Z 614.955,A -85,B 0,C 180,E1 -14516.869,E2 -14516.869} C_VEL
LIN {X 0,Y 337.432,Z 604.753,A -85,B 0,C 180,E1 -14518.982,E2 -14518.982} C_VEL
LIN {X 0,Y 333.648,Z 588.926,A -85,B 0,C 180,E1 -14522.442,E2 -14522.442} C_VEL
LIN {X 0,Y 333.676,Z 588.922,A -85,B 0,C 180,E1 -14526.138,E2 -14526.138} C_VEL
LIN {X 0,Y 333.67,Z 588.918,A -85,B 0,C 180,E1 -14529.188,E2 -14529.188} C_VEL
LIN {X 0,Y 333.673,Z 588.917,A -85,B 0,C 180,E1 -14532.507,E2 -14532.507} C_VEL
LIN {X 0,Y 333.666,Z 588.914,A -85,B 0,C 180,E1 -14535.966,E2 -14535.966} C_VEL
LIN {X 0,Y 333.698,Z 588.914,A -85,B 0,C 180,E1 -14539.304,E2 -14539.304} C_VEL
LIN {X 0,Y 333.663,Z 588.92,A -85,B 0,C 180,E1 -14543.166,E2 -14543.166} C_VEL
LIN {X 0,Y 333.636,Z 588.922,A -85,B 0,C 180,E1 -14546.791,E2 -14546.791} C_VEL
LIN {X 0,Y 333.699,Z 588.913,A -85,B 0,C 180,E1 -14549.709,E2 -14549.709} C_VEL
LIN {X 0,Y 333.738,Z 588.904,A -85,B 0,C 180,E1 -14552.401,E2 -14552.401} C_VEL
LIN {X 0,Y 333.72,Z 588.911,A -85,B 0,C 180,E1 -14555.09,E2 -14555.09} C_VEL
LIN {X 0,Y 333.673,Z 588.917,A -85,B 0,C 180,E1 -14559.019,E2 -14559.019} C_VEL
LIN {X 0,Y 333.786,Z 588.904,A -85,B 0,C 180,E1 -14561.589,E2 -14561.589} C_VEL
LIN {X 0,Y 333.801,Z 588.896,A -85,B 0,C 180,E1 -14565.576,E2 -14565.576} C_VEL
LIN {X 0,Y 333.826,Z 588.894,A -85,B 0,C 180,E1 -14569.078,E2 -14569.078} C_VEL
LIN {X 0,Y 334,Z 588.87,A -85,B 0,C 180,E1 -14572.747,E2 -14572.747} C_VEL
LIN {X 0,Y 333.808,Z 588.902,A -85,B 0,C 180,E1 -14575.169,E2 -14575.169} C_VEL
LIN {X 0,Y 334.1,Z 588.851,A -85,B 0,C 180,E1 -14577.589,E2 -14577.589} C_VEL
LIN {X 0,Y 334.24,Z 588.84,A -85,B 0,C 180,E1 -14580,E2 -14580} C_VEL
LIN {X 0,Y 334.124,Z 588.866,A -85,B 0,C 180,E1 -14582.411,E2 -14582.411} C_VEL
LIN {X 0,Y 334.006,Z 588.871,A -85,B 0,C 180,E1 -14587.253,E2 -14587.253} C_VEL
LIN {X 0,Y 333.826,Z 588.893,A -85,B 0,C 180,E1 -14590.922,E2 -14590.922} C_VEL
LIN {X 0,Y 333.801,Z 588.9,A -85,B 0,C 180,E1 -14594.635,E2 -14594.635} C_VEL
LIN {X 0,Y 333.789,Z 588.892,A -85,B 0,C 180,E1 -14598.655,E2 -14598.655} C_VEL
LIN {X 0,Y 333.685,Z 588.919,A -85,B 0,C 180,E1 -14602.279,E2 -14602.279} C_VEL
LIN {X 0,Y 333.729,Z 588.909,A -85,B 0,C 180,E1 -14606.247,E2 -14606.247} C_VEL
LIN {X 0,Y 333.706,Z 588.909,A -85,B 0,C 180,E1 -14608.973,E2 -14608.973} C_VEL
LIN {X 0,Y 333.646,Z 588.925,A -85,B 0,C 180,E1 -14612.59,E2 -14612.59} C_VEL
LIN {X 0,Y 333.671,Z 588.92,A -85,B 0,C 180,E1 -14616.14,E2 -14616.14} C_VEL
LIN {X 0,Y 333.668,Z 588.922,A -85,B 0,C 180,E1 -14619.19,E2 -14619.19} C_VEL
LIN {X 0,Y 333.662,Z 588.893,A -85,B 0,C 180,E1 -14622.507,E2 -14622.507} C_VEL
LIN {X 0,Y 333.619,Z 588.924,A -85,B 0,C 180,E1 -14625.96,E2 -14625.96} C_VEL
LIN {X 0,Y 333.645,Z 588.919,A -85,B 0,C 180,E1 -14629.316,E2 -14629.316} C_VEL
LIN {X 0,Y 333.685,Z 589.032,A -85,B 0,C 180,E1 -14632.7,E2 -14632.7} C_VEL
LIN {X 0,Y 334.721,Z 591.855,A -85,B 0,C 180,E1 -14632.87,E2 -14632.87} C_VEL
LIN {X 0,Y 342.003,Z 605.85,A -85,B 0,C 180,E1 -14633.887,E2 -14633.887} C_VEL
LIN {X 0,Y 346.749,Z 616.062,A -85,B 0,C 180,E1 -14634.544,E2 -14634.544} C_VEL
LIN {X 0,Y 345.155,Z 684.813,A -85,B 0,C 180,E1 -14635.993,E2 -14635.993} C_VEL
LIN {X 0,Y 344.727,Z 698.226,A -85,B 0,C 180,E1 -14636.472,E2 -14636.472} C_VEL
LIN {X 0,Y 344.099,Z 709.845,A -85,B 0,C 180,E1 -14637.099,E2 -14637.099} C_VEL
LIN {X 0,Y 343.039,Z 722.054,A -85,B 0,C 180,E1 -14637.988,E2 -14637.988} C_VEL
LIN {X 0,Y 341.817,Z 733.299,A -85,B 0,C 180,E1 -14639.069,E2 -14639.069} C_VEL
LIN {X 0,Y 340.48,Z 743.539,A -85,B 0,C 180,E1 -14640.305,E2 -14640.305} C_VEL
LIN {X 0,Y 339.264,Z 751.917,A -85,B 0,C 180,E1 -14641.547,E2 -14641.547} C_VEL
LIN {X 0,Y 337.861,Z 761.273,A -85,B 0,C 180,E1 -14643.261,E2 -14643.261} C_VEL
LIN {X 0,Y 336.528,Z 768.823,A -85,B 0,C 180,E1 -14644.983,E2 -14644.983} C_VEL
LIN {X 0,Y 335.25,Z 775.975,A -85,B 0,C 180,E1 -14647.042,E2 -14647.042} C_VEL
LIN {X 0,Y 334.309,Z 781.29,A -85,B 0,C 180,E1 -14649.061,E2 -14649.061} C_VEL
LIN {X 0,Y 333.582,Z 785.125,A -85,B 0,C 180,E1 -14651.004,E2 -14651.004} C_VEL
LIN {X 0,Y 333.083,Z 787.675,A -85,B 0,C 180,E1 -14652.819,E2 -14652.819} C_VEL
LIN {X 0,Y 332.808,Z 788.9,A -85,B 0,C 180,E1 -14654.067,E2 -14654.067} C_VEL
LIN {X 0,Y 332.628,Z 789.704,A -85,B 0,C 180,E1 -14655.313,E2 -14655.313} C_VEL
LIN {X 0,Y 332.529,Z 790.058,A -85,B 0,C 180,E1 -14656.557,E2 -14656.557} C_VEL
LIN {X 0,Y 332.473,Z 790.023,A -85,B 0,C 180,E1 -14657.797,E2 -14657.797} C_VEL
LIN {X 0,Y 332.416,Z 789.606,A -85,B 0,C 180,E1 -14659.031,E2 -14659.031} C_VEL
LIN {X 0,Y 332.479,Z 788.742,A -85,B 0,C 180,E1 -14660.264,E2 -14660.264} C_VEL
LIN {X 0,Y 332.574,Z 787.477,A -85,B 0,C 180,E1 -14661.494,E2 -14661.494} C_VEL
LIN {X 0,Y 332.81,Z 785.392,A -85,B 0,C 180,E1 -14662.983,E2 -14662.983} C_VEL
LIN {X 0,Y 333.226,Z 781.1,A -85,B 0,C 180,E1 -14665.161,E2 -14665.161} C_VEL
LIN {X 0,Y 333.648,Z 776.314,A -85,B 0,C 180,E1 -14666.981,E2 -14666.981} C_VEL
LIN {X 0,Y 334.336,Z 770.268,A -85,B 0,C 180,E1 -14668.796,E2 -14668.796} C_VEL
LIN {X 0,Y 335.141,Z 762.723,A -85,B 0,C 180,E1 -14670.601,E2 -14670.601} C_VEL
LIN {X 0,Y 336.255,Z 753.267,A -85,B 0,C 180,E1 -14672.396,E2 -14672.396} C_VEL
LIN {X 0,Y 337.282,Z 743.504,A -85,B 0,C 180,E1 -14673.883,E2 -14673.883} C_VEL
LIN {X 0,Y 338.28,Z 732.533,A -85,B 0,C 180,E1 -14675.215,E2 -14675.215} C_VEL
LIN {X 0,Y 339.277,Z 721.468,A -85,B 0,C 180,E1 -14676.273,E2 -14676.273} C_VEL
LIN {X 0,Y 340.014,Z 710.006,A -85,B 0,C 180,E1 -14677.124,E2 -14677.124} C_VEL
LIN {X 0,Y 340.57,Z 696.873,A -85,B 0,C 180,E1 -14677.831,E2 -14677.831} C_VEL
LIN {X 0,Y 340.929,Z 684.592,A -85,B 0,C 180,E1 -14678.261,E2 -14678.261} C_VEL
LIN {X 0,Y 342.2,Z 610.829,A -85,B 0,C 180,E1 -14679.81,E2 -14679.81} C_VEL
LIN {X 0,Y 333.963,Z 589.647,A -85,B 0,C 180,E1 -14680.764,E2 -14680.764} C_VEL
LIN {X 0,Y 333.838,Z 588.899,A -85,B 0,C 180,E1 -14680.806,E2 -14680.806} C_VEL
LIN {X 0,Y 333.81,Z 588.904,A -85,B 0,C 180,E1 -14684.634,E2 -14684.634} C_VEL
LIN {X 0,Y 333.798,Z 588.905,A -85,B 0,C 180,E1 -14688.655,E2 -14688.655} C_VEL
LIN {X 0,Y 333.691,Z 588.917,A -85,B 0,C 180,E1 -14692.808,E2 -14692.808} C_VEL
LIN {X 0,Y 336.316,Z 595.799,A -85,B 0,C 180,E1 -14693.151,E2 -14693.151} C_VEL
LIN {X 0,Y 342.912,Z 612.321,A -85,B 0,C 180,E1 -14693.957,E2 -14693.957} C_VEL
LIN {X 0,Y 342.867,Z 616.697,A -85,B 0,C 180,E1 -14694.06,E2 -14694.06} C_VEL
LIN {X 0,Y 342.081,Z 622.525,A -85,B 0,C 180,E1 -14694.156,E2 -14694.156} C_VEL
LIN {X 0,Y 336.205,Z 641.457,A -85,B 0,C 180,E1 -14694.27,E2 -14694.27} C_VEL
LIN {X 0,Y 335.376,Z 647.287,A -85,B 0,C 180,E1 -14694.364,E2 -14694.364} C_VEL
LIN {X 0,Y 334.455,Z 687.48,A -85,B 0,C 180,E1 -14695.327,E2 -14695.327} C_VEL
LIN {X 0,Y 334.023,Z 700.807,A -85,B 0,C 180,E1 -14695.886,E2 -14695.886} C_VEL
LIN {X 0,Y 333.344,Z 712.875,A -85,B 0,C 180,E1 -14696.616,E2 -14696.616} C_VEL
LIN {X 0,Y 332.435,Z 724.814,A -85,B 0,C 180,E1 -14697.585,E2 -14697.585} C_VEL
LIN {X 0,Y 331.413,Z 736.752,A -85,B 0,C 180,E1 -14698.844,E2 -14698.844} C_VEL
LIN {X 0,Y 330.345,Z 747.126,A -85,B 0,C 180,E1 -14700.215,E2 -14700.215} C_VEL
LIN {X 0,Y 329.24,Z 756.747,A -85,B 0,C 180,E1 -14701.802,E2 -14701.802} C_VEL
LIN {X 0,Y 328.183,Z 765.443,A -85,B 0,C 180,E1 -14703.575,E2 -14703.575} C_VEL
LIN {X 0,Y 327.308,Z 772.757,A -85,B 0,C 180,E1 -14705.432,E2 -14705.432} C_VEL
LIN {X 0,Y 326.698,Z 778.457,A -85,B 0,C 180,E1 -14707.254,E2 -14707.254} C_VEL
LIN {X 0,Y 326.146,Z 783.077,A -85,B 0,C 180,E1 -14709.127,E2 -14709.127} C_VEL
LIN {X 0,Y 325.756,Z 786.528,A -85,B 0,C 180,E1 -14710.965,E2 -14710.965} C_VEL
LIN {X 0,Y 325.474,Z 788.96,A -85,B 0,C 180,E1 -14712.763,E2 -14712.763} C_VEL
LIN {X 0,Y 325.316,Z 790.469,A -85,B 0,C 180,E1 -14714.527,E2 -14714.527} C_VEL
LIN {X 0,Y 325.314,Z 791.139,A -85,B 0,C 180,E1 -14716.265,E2 -14716.265} C_VEL
LIN {X 0,Y 325.438,Z 791.039,A -85,B 0,C 180,E1 -14717.974,E2 -14717.974} C_VEL
LIN {X 0,Y 325.653,Z 790.218,A -85,B 0,C 180,E1 -14719.651,E2 -14719.651} C_VEL
LIN {X 0,Y 326.242,Z 787.584,A -85,B 0,C 180,E1 -14722.109,E2 -14722.109} C_VEL
LIN {X 0,Y 326.976,Z 783.345,A -85,B 0,C 180,E1 -14724.526,E2 -14724.526} C_VEL
LIN {X 0,Y 327.921,Z 777.904,A -85,B 0,C 180,E1 -14726.702,E2 -14726.702} C_VEL
LIN {X 0,Y 329.069,Z 771.444,A -85,B 0,C 180,E1 -14728.679,E2 -14728.679} C_VEL
LIN {X 0,Y 330.213,Z 764.612,A -85,B 0,C 180,E1 -14730.342,E2 -14730.342} C_VEL
LIN {X 0,Y 331.549,Z 756.013,A -85,B 0,C 180,E1 -14732.031,E2 -14732.031} C_VEL
LIN {X 0,Y 332.961,Z 746.494,A -85,B 0,C 180,E1 -14733.538,E2 -14733.538} C_VEL
LIN {X 0,Y 334.3,Z 735.865,A -85,B 0,C 180,E1 -14734.896,E2 -14734.896} C_VEL
LIN {X 0,Y 335.509,Z 724.282,A -85,B 0,C 180,E1 -14736.055,E2 -14736.055} C_VEL
LIN {X 0,Y 336.664,Z 711.391,A -85,B 0,C 180,E1 -14737.036,E2 -14737.036} C_VEL
LIN {X 0,Y 337.323,Z 698.36,A -85,B 0,C 180,E1 -14737.752,E2 -14737.752} C_VEL
LIN {X 0,Y 337.747,Z 685.912,A -85,B 0,C 180,E1 -14738.2,E2 -14738.2} C_VEL
LIN {X 0,Y 339.873,Z 617.197,A -85,B 0,C 180,E1 -14739.853,E2 -14739.853} C_VEL
LIN {X 0,Y 332.222,Z 601.041,A -85,B 0,C 180,E1 -14741.042,E2 -14741.042} C_VEL
LIN {X 0,Y 327.917,Z 592.892,A -85,B 0,C 180,E1 -14741.733,E2 -14741.733} C_VEL
LIN {X 0,Y 326.733,Z 589.943,A -85,B 0,C 180,E1 -14741.948,E2 -14741.948} C_VEL
LIN {X 0,Y 326.756,Z 589.785,A -85,B 0,C 180,E1 -14745.433,E2 -14745.433} C_VEL
LIN {X 0,Y 326.766,Z 589.782,A -85,B 0,C 180,E1 -14748.839,E2 -14748.839} C_VEL
LIN {X 0,Y 326.973,Z 589.754,A -85,B 0,C 180,E1 -14752.59,E2 -14752.59} C_VEL
LIN {X 0,Y 326.775,Z 589.778,A -85,B 0,C 180,E1 -14755.065,E2 -14755.065} C_VEL
LIN {X 0,Y 327.041,Z 589.743,A -85,B 0,C 180,E1 -14757.537,E2 -14757.537} C_VEL
LIN {X 0,Y 327.21,Z 589.724,A -85,B 0,C 180,E1 -14760,E2 -14760} C_VEL
LIN {X 0,Y 327.041,Z 589.747,A -85,B 0,C 180,E1 -14762.463,E2 -14762.463} C_VEL
LIN {X 0,Y 326.987,Z 589.75,A -85,B 0,C 180,E1 -14766.169,E2 -14766.169} C_VEL
LIN {X 0,Y 326.907,Z 589.762,A -85,B 0,C 180,E1 -14768.655,E2 -14768.655} C_VEL
LIN {X 0,Y 326.731,Z 589.78,A -85,B 0,C 180,E1 -14772.421,E2 -14772.421} C_VEL
LIN {X 0,Y 326.747,Z 589.779,A -85,B 0,C 180,E1 -14774.958,E2 -14774.958} C_VEL
LIN {X 0,Y 326.727,Z 589.782,A -85,B 0,C 180,E1 -14778.839,E2 -14778.839} C_VEL
LIN {X 0,Y 326.614,Z 589.797,A -85,B 0,C 180,E1 -14782.788,E2 -14782.788} C_VEL
LIN {X 0,Y 326.684,Z 589.791,A -85,B 0,C 180,E1 -14785.484,E2 -14785.484} C_VEL
LIN {X 0,Y 326.655,Z 589.794,A -85,B 0,C 180,E1 -14789.66,E2 -14789.66} C_VEL
LIN {X 0,Y 326.603,Z 589.797,A -85,B 0,C 180,E1 -14794.02,E2 -14794.02} C_VEL
LIN {X 0,Y 326.625,Z 589.799,A -85,B 0,C 180,E1 -14797.24,E2 -14797.24} C_VEL
LIN {X 0,Y 326.631,Z 589.798,A -85,B 0,C 180,E1 -14800.203,E2 -14800.203} C_VEL
LIN {X 0,Y 326.615,Z 589.8,A -85,B 0,C 180,E1 -14803.517,E2 -14803.517} C_VEL
LIN {X 0,Y 326.614,Z 589.803,A -85,B 0,C 180,E1 -14807.021,E2 -14807.021} C_VEL
LIN {X 0,Y 326.641,Z 589.798,A -85,B 0,C 180,E1 -14811.395,E2 -14811.395} C_VEL
LIN {X 0,Y 326.664,Z 589.945,A -85,B 0,C 180,E1 -14813.631,E2 -14813.631} C_VEL
LIN {X 0,Y 329.047,Z 599.073,A -85,B 0,C 180,E1 -14816.407,E2 -14816.407} C_VEL
LIN {X 0,Y 331.508,Z 609.736,A -85,B 0,C 180,E1 -14819.417,E2 -14819.417} C_VEL
LIN {X 0,Y 332.913,Z 618.263,A -85,B 0,C 180,E1 -14821.642,E2 -14821.642} C_VEL
LIN {X 0,Y 331.252,Z 630.368,A -85,B 0,C 180,E1 -14824.388,E2 -14824.388} C_VEL
LIN {X 0,Y 335.59,Z 655.652,A -85,B 0,C 180,E1 -14825.505,E2 -14825.505} C_VEL
LIN {X 0,Y 338.397,Z 681.244,A -85,B 0,C 180,E1 -14826.445,E2 -14826.445} C_VEL
LIN {X 0,Y 336.538,Z 742.237,A -85,B 0,C 180,E1 -14827.921,E2 -14827.921} C_VEL
LIN {X 0,Y 335.565,Z 756.141,A -85,B 0,C 180,E1 -14828.5,E2 -14828.5} C_VEL
LIN {X 0,Y 334.369,Z 768.164,A -85,B 0,C 180,E1 -14829.226,E2 -14829.226} C_VEL
LIN {X 0,Y 332.785,Z 780.755,A -85,B 0,C 180,E1 -14830.252,E2 -14830.252} C_VEL
LIN {X 0,Y 331.303,Z 792.075,A -85,B 0,C 180,E1 -14831.446,E2 -14831.446} C_VEL
LIN {X 0,Y 329.778,Z 802.346,A -85,B 0,C 180,E1 -14832.801,E2 -14832.801} C_VEL
LIN {X 0,Y 328.42,Z 812.762,A -85,B 0,C 180,E1 -14834.532,E2 -14834.532} C_VEL
LIN {X 0,Y 327.055,Z 821.539,A -85,B 0,C 180,E1 -14836.328,E2 -14836.328} C_VEL
LIN {X 0,Y 326.141,Z 828.799,A -85,B 0,C 180,E1 -14838.187,E2 -14838.187} C_VEL
LIN {X 0,Y 325.553,Z 834.657,A -85,B 0,C 180,E1 -14840.055,E2 -14840.055} C_VEL
LIN {X 0,Y 325.277,Z 839.307,A -85,B 0,C 180,E1 -14841.927,E2 -14841.927} C_VEL
LIN {X 0,Y 325.193,Z 842.863,A -85,B 0,C 180,E1 -14843.797,E2 -14843.797} C_VEL
LIN {X 0,Y 325.184,Z 844.656,A -85,B 0,C 180,E1 -14845.041,E2 -14845.041} C_VEL
LIN {X 0,Y 325.185,Z 846.032,A -85,B 0,C 180,E1 -14846.283,E2 -14846.283} C_VEL
LIN {X 0,Y 325.389,Z 846.981,A -85,B 0,C 180,E1 -14847.524,E2 -14847.524} C_VEL
LIN {X 0,Y 325.415,Z 847.476,A -85,B 0,C 180,E1 -14848.763,E2 -14848.763} C_VEL
LIN {X 0,Y 325.514,Z 847.572,A -85,B 0,C 180,E1 -14850,E2 -14850} C_VEL
LIN {X 0,Y 325.451,Z 847.247,A -85,B 0,C 180,E1 -14851.237,E2 -14851.237} C_VEL
LIN {X 0,Y 325.416,Z 846.478,A -85,B 0,C 180,E1 -14852.476,E2 -14852.476} C_VEL
LIN {X 0,Y 325.236,Z 843.676,A -85,B 0,C 180,E1 -14854.958,E2 -14854.958} C_VEL
LIN {X 0,Y 325.17,Z 841.188,A -85,B 0,C 180,E1 -14856.765,E2 -14856.765} C_VEL
LIN {X 0,Y 325.347,Z 837.498,A -85,B 0,C 180,E1 -14858.697,E2 -14858.697} C_VEL
LIN {X 0,Y 325.727,Z 832.806,A -85,B 0,C 180,E1 -14860.568,E2 -14860.568} C_VEL
LIN {X 0,Y 326.646,Z 825.745,A -85,B 0,C 180,E1 -14862.74,E2 -14862.74} C_VEL
LIN {X 0,Y 327.767,Z 818.144,A -85,B 0,C 180,E1 -14864.592,E2 -14864.592} C_VEL
LIN {X 0,Y 328.842,Z 810.395,A -85,B 0,C 180,E1 -14866.131,E2 -14866.131} C_VEL
LIN {X 0,Y 330.335,Z 800.958,A -85,B 0,C 180,E1 -14867.648,E2 -14867.648} C_VEL
LIN {X 0,Y 331.97,Z 790.511,A -85,B 0,C 180,E1 -14868.995,E2 -14868.995} C_VEL
LIN {X 0,Y 333.55,Z 778.901,A -85,B 0,C 180,E1 -14870.183,E2 -14870.183} C_VEL
LIN {X 0,Y 335.098,Z 766.503,A -85,B 0,C 180,E1 -14871.129,E2 -14871.129} C_VEL
LIN {X 0,Y 336.323,Z 753.481,A -85,B 0,C 180,E1 -14871.852,E2 -14871.852} C_VEL
LIN {X 0,Y 337.163,Z 740.879,A -85,B 0,C 180,E1 -14872.302,E2 -14872.302} C_VEL
LIN {X 0,Y 338.56,Z 678.116,A -85,B 0,C 180,E1 -14873.681,E2 -14873.681} C_VEL
LIN {X 0,Y 335.51,Z 649.824,A -85,B 0,C 180,E1 -14874.622,E2 -14874.622} C_VEL
LIN {X 0,Y 331.74,Z 623.694,A -85,B 0,C 180,E1 -14875.615,E2 -14875.615} C_VEL
LIN {X 0,Y 332.511,Z 615.684,A -85,B 0,C 180,E1 -14877.14,E2 -14877.14} C_VEL
LIN {X 0,Y 329.891,Z 603.732,A -85,B 0,C 180,E1 -14879.69,E2 -14879.69} C_VEL
LIN {X 0,Y 326.596,Z 589.803,A -85,B 0,C 180,E1 -14882.83,E2 -14882.83} C_VEL
LIN {X 0,Y 326.612,Z 589.802,A -85,B 0,C 180,E1 -14885.519,E2 -14885.519} C_VEL
LIN {X 0,Y 326.633,Z 589.794,A -85,B 0,C 180,E1 -14889.231,E2 -14889.231} C_VEL
LIN {X 0,Y 326.607,Z 589.8,A -85,B 0,C 180,E1 -14893.517,E2 -14893.517} C_VEL
LIN {X 0,Y 326.624,Z 589.797,A -85,B 0,C 180,E1 -14897.018,E2 -14897.018} C_VEL
LIN {X 0,Y 326.641,Z 589.787,A -85,B 0,C 180,E1 -14900.765,E2 -14900.765} C_VEL
LIN {X 0,Y 326.608,Z 589.789,A -85,B 0,C 180,E1 -14904.48,E2 -14904.48} C_VEL
LIN {X 0,Y 326.61,Z 589.798,A -85,B 0,C 180,E1 -14907.456,E2 -14907.456} C_VEL
LIN {X 0,Y 326.656,Z 589.781,A -85,B 0,C 180,E1 -14910.34,E2 -14910.34} C_VEL
LIN {X 0,Y 326.684,Z 589.792,A -85,B 0,C 180,E1 -14914.516,E2 -14914.516} C_VEL
LIN {X 0,Y 326.639,Z 589.784,A -85,B 0,C 180,E1 -14918.545,E2 -14918.545} C_VEL
LIN {X 0,Y 326.738,Z 589.782,A -85,B 0,C 180,E1 -14921.177,E2 -14921.177} C_VEL
LIN {X 0,Y 326.756,Z 589.773,A -85,B 0,C 180,E1 -14925.433,E2 -14925.433} C_VEL
LIN {X 0,Y 326.762,Z 589.776,A -85,B 0,C 180,E1 -14928.839,E2 -14928.839} C_VEL
LIN {X 0,Y 326.952,Z 589.745,A -85,B 0,C 180,E1 -14932.59,E2 -14932.59} C_VEL
LIN {X 0,Y 326.775,Z 589.779,A -85,B 0,C 180,E1 -14935.065,E2 -14935.065} C_VEL
LIN {X 0,Y 327.041,Z 589.731,A -85,B 0,C 180,E1 -14937.537,E2 -14937.537} C_VEL
LIN {X 0,Y 327.192,Z 589.717,A -85,B 0,C 180,E1 -14940,E2 -14940} C_VEL
LIN {X 0,Y 327.061,Z 589.746,A -85,B 0,C 180,E1 -14942.463,E2 -14942.463} C_VEL
LIN {X 0,Y 326.957,Z 589.74,A -85,B 0,C 180,E1 -14946.615,E2 -14946.615} C_VEL
LIN {X 0,Y 326.907,Z 589.763,A -85,B 0,C 180,E1 -14948.655,E2 -14948.655} C_VEL
LIN {X 0,Y 326.726,Z 589.768,A -85,B 0,C 180,E1 -14952.422,E2 -14952.422} C_VEL
LIN {X 0,Y 326.747,Z 589.782,A -85,B 0,C 180,E1 -14954.958,E2 -14954.958} C_VEL
LIN {X 0,Y 326.726,Z 589.771,A -85,B 0,C 180,E1 -14958.838,E2 -14958.838} C_VEL
LIN {X 0,Y 326.613,Z 589.799,A -85,B 0,C 180,E1 -14962.788,E2 -14962.788} C_VEL
LIN {X 0,Y 326.684,Z 589.782,A -85,B 0,C 180,E1 -14965.484,E2 -14965.484} C_VEL
LIN {X 0,Y 326.656,Z 589.783,A -85,B 0,C 180,E1 -14969.66,E2 -14969.66} C_VEL
LIN {X 0,Y 326.618,Z 589.799,A -85,B 0,C 180,E1 -14972.948,E2 -14972.948} C_VEL
LIN {X 0,Y 326.627,Z 589.799,A -85,B 0,C 180,E1 -14977.047,E2 -14977.047} C_VEL
LIN {X 0,Y 326.6,Z 589.795,A -85,B 0,C 180,E1 -14980.208,E2 -14980.208} C_VEL
LIN {X 0,Y 326.588,Z 589.784,A -85,B 0,C 180,E1 -14983.521,E2 -14983.521} C_VEL
LIN {X 0,Y 326.579,Z 589.788,A -85,B 0,C 180,E1 -14987.028,E2 -14987.028} C_VEL
LIN {X 0,Y 326.609,Z 589.797,A -85,B 0,C 180,E1 -14990.774,E2 -14990.774} C_VEL
LIN {X 0,Y 326.628,Z 589.981,A -85,B 0,C 180,E1 -14992.015,E2 -14992.015} C_VEL
LIN {X 0,Y 327.812,Z 592.961,A -85,B 0,C 180,E1 -14992.211,E2 -14992.211} C_VEL
LIN {X 0,Y 336.24,Z 609.024,A -85,B 0,C 180,E1 -14993.43,E2 -14993.43} C_VEL
LIN {X 0,Y 340.443,Z 618.317,A -85,B 0,C 180,E1 -14994.039,E2 -14994.039} C_VEL
LIN {X 0,Y 338.812,Z 684.628,A -85,B 0,C 180,E1 -14995.457,E2 -14995.457} C_VEL
LIN {X 0,Y 338.409,Z 697.332,A -85,B 0,C 180,E1 -14995.895,E2 -14995.895} C_VEL
LIN {X 0,Y 337.792,Z 708.91,A -85,B 0,C 180,E1 -14996.507,E2 -14996.507} C_VEL
LIN {X 0,Y 336.812,Z 720.406,A -85,B 0,C 180,E1 -14997.323,E2 -14997.323} C_VEL
LIN {X 0,Y 335.54,Z 732.235,A -85,B 0,C 180,E1 -14998.425,E2 -14998.425} C_VEL
LIN {X 0,Y 334.107,Z 742.765,A -85,B 0,C 180,E1 -14999.68,E2 -14999.68} C_VEL
LIN {X 0,Y 332.494,Z 753.327,A -85,B 0,C 180,E1 -15001.258,E2 -15001.258} C_VEL
LIN {X 0,Y 331.232,Z 761.394,A -85,B 0,C 180,E1 -15002.77,E2 -15002.77} C_VEL
LIN {X 0,Y 329.872,Z 768.709,A -85,B 0,C 180,E1 -15004.442,E2 -15004.442} C_VEL
LIN {X 0,Y 328.816,Z 774.427,A -85,B 0,C 180,E1 -15006.041,E2 -15006.041} C_VEL
LIN {X 0,Y 327.744,Z 779.925,A -85,B 0,C 180,E1 -15007.96,E2 -15007.96} C_VEL
LIN {X 0,Y 326.924,Z 784.158,A -85,B 0,C 180,E1 -15009.882,E2 -15009.882} C_VEL
LIN {X 0,Y 326.452,Z 786.588,A -85,B 0,C 180,E1 -15011.308,E2 -15011.308} C_VEL
LIN {X 0,Y 325.816,Z 789.348,A -85,B 0,C 180,E1 -15013.715,E2 -15013.715} C_VEL
LIN {X 0,Y 325.607,Z 790.216,A -85,B 0,C 180,E1 -15014.989,E2 -15014.989} C_VEL
LIN {X 0,Y 325.478,Z 790.653,A -85,B 0,C 180,E1 -15016.332,E2 -15016.332} C_VEL
LIN {X 0,Y 325.341,Z 790.287,A -85,B 0,C 180,E1 -15018.79,E2 -15018.79} C_VEL
LIN {X 0,Y 325.383,Z 789.513,A -85,B 0,C 180,E1 -15020.05,E2 -15020.05} C_VEL
LIN {X 0,Y 325.495,Z 788.293,A -85,B 0,C 180,E1 -15021.307,E2 -15021.307} C_VEL
LIN {X 0,Y 325.74,Z 786.071,A -85,B 0,C 180,E1 -15022.967,E2 -15022.967} C_VEL
LIN {X 0,Y 326.146,Z 782.11,A -85,B 0,C 180,E1 -15025.055,E2 -15025.055} C_VEL
LIN {X 0,Y 326.571,Z 777.43,A -85,B 0,C 180,E1 -15026.916,E2 -15026.916} C_VEL
LIN {X 0,Y 327.254,Z 771.502,A -85,B 0,C 180,E1 -15028.769,E2 -15028.769} C_VEL
LIN {X 0,Y 328.073,Z 764.143,A -85,B 0,C 180,E1 -15030.614,E2 -15030.614} C_VEL
LIN {X 0,Y 329.197,Z 754.866,A -85,B 0,C 180,E1 -15032.447,E2 -15032.447} C_VEL
LIN {X 0,Y 330.245,Z 745.336,A -85,B 0,C 180,E1 -15033.966,E2 -15033.966} C_VEL
LIN {X 0,Y 331.267,Z 734.703,A -85,B 0,C 180,E1 -15035.326,E2 -15035.326} C_VEL
LIN {X 0,Y 332.402,Z 722.65,A -85,B 0,C 180,E1 -15036.526,E2 -15036.526} C_VEL
LIN {X 0,Y 333.18,Z 711.498,A -85,B 0,C 180,E1 -15037.386,E2 -15037.386} C_VEL
LIN {X 0,Y 333.75,Z 698.423,A -85,B 0,C 180,E1 -15038.123,E2 -15038.123} C_VEL
LIN {X 0,Y 334.149,Z 684.966,A -85,B 0,C 180,E1 -15038.613,E2 -15038.613} C_VEL
LIN {X 0,Y 335.393,Z 612.2,A -85,B 0,C 180,E1 -15040.173,E2 -15040.173} C_VEL
LIN {X 0,Y 326.949,Z 590.593,A -85,B 0,C 180,E1 -15041.179,E2 -15041.179} C_VEL
LIN {X 0,Y 326.768,Z 589.78,A -85,B 0,C 180,E1 -15041.239,E2 -15041.239} C_VEL
LIN {X 0,Y 326.756,Z 589.781,A -85,B 0,C 180,E1 -15044.957,E2 -15044.957} C_VEL
LIN {X 0,Y 326.733,Z 589.785,A -85,B 0,C 180,E1 -15048.837,E2 -15048.837} C_VEL
LIN {X 0,Y 326.666,Z 589.879,A -85,B 0,C 180,E1 -15052.372,E2 -15052.372} C_VEL
LIN {X 0,Y 329.25,Z 596.634,A -85,B 0,C 180,E1 -15052.719,E2 -15052.719} C_VEL
LIN {X 0,Y 336.213,Z 614.012,A -85,B 0,C 180,E1 -15053.598,E2 -15053.598} C_VEL
LIN {X 0,Y 335.376,Z 647.287,A -85,B 0,C 180,E1 -15054.364,E2 -15054.364} C_VEL
LIN {X 0,Y 334.549,Z 653.115,A -85,B 0,C 180,E1 -15054.457,E2 -15054.457} C_VEL
LIN {X 0,Y 328.692,Z 672.041,A -85,B 0,C 180,E1 -15054.588,E2 -15054.588} C_VEL
LIN {X 0,Y 327.898,Z 677.867,A -85,B 0,C 180,E1 -15054.688,E2 -15054.688} C_VEL
LIN {X 0,Y 327.577,Z 692.682,A -85,B 0,C 180,E1 -15055.129,E2 -15055.129} C_VEL
LIN {X 0,Y 327.079,Z 704.896,A -85,B 0,C 180,E1 -15055.727,E2 -15055.727} C_VEL
LIN {X 0,Y 326.215,Z 717.857,A -85,B 0,C 180,E1 -15056.614,E2 -15056.614} C_VEL
LIN {X 0,Y 325.224,Z 730.114,A -85,B 0,C 180,E1 -15057.736,E2 -15057.736} C_VEL
LIN {X 0,Y 324.14,Z 741.065,A -85,B 0,C 180,E1 -15059.02,E2 -15059.02} C_VEL
LIN {X 0,Y 322.957,Z 751.696,A -85,B 0,C 180,E1 -15060.575,E2 -15060.575} C_VEL
LIN {X 0,Y 322.054,Z 759.558,A -85,B 0,C 180,E1 -15061.99,E2 -15061.99} C_VEL
LIN {X 0,Y 321.049,Z 767.445,A -85,B 0,C 180,E1 -15063.711,E2 -15063.711} C_VEL
LIN {X 0,Y 320.134,Z 774.69,A -85,B 0,C 180,E1 -15065.681,E2 -15065.681} C_VEL
LIN {X 0,Y 319.505,Z 780.384,A -85,B 0,C 180,E1 -15067.639,E2 -15067.639} C_VEL
LIN {X 0,Y 318.952,Z 785.047,A -85,B 0,C 180,E1 -15069.716,E2 -15069.716} C_VEL
LIN {X 0,Y 318.582,Z 787.903,A -85,B 0,C 180,E1 -15071.437,E2 -15071.437} C_VEL
LIN {X 0,Y 318.335,Z 790.036,A -85,B 0,C 180,E1 -15073.235,E2 -15073.235} C_VEL
LIN {X 0,Y 318.229,Z 791.339,A -85,B 0,C 180,E1 -15075.032,E2 -15075.032} C_VEL
LIN {X 0,Y 318.267,Z 791.838,A -85,B 0,C 180,E1 -15076.8,E2 -15076.8} C_VEL
LIN {X 0,Y 318.453,Z 791.51,A -85,B 0,C 180,E1 -15078.619,E2 -15078.619} C_VEL
LIN {X 0,Y 318.764,Z 790.284,A -85,B 0,C 180,E1 -15080.502,E2 -15080.502} C_VEL
LIN {X 0,Y 319.28,Z 788.102,A -85,B 0,C 180,E1 -15082.412,E2 -15082.412} C_VEL
LIN {X 0,Y 319.882,Z 784.82,A -85,B 0,C 180,E1 -15084.379,E2 -15084.379} C_VEL
LIN {X 0,Y 320.716,Z 780.302,A -85,B 0,C 180,E1 -15086.376,E2 -15086.376} C_VEL
LIN {X 0,Y 321.864,Z 774.294,A -85,B 0,C 180,E1 -15088.396,E2 -15088.396} C_VEL
LIN {X 0,Y 323.239,Z 766.566,A -85,B 0,C 180,E1 -15090.421,E2 -15090.421} C_VEL
LIN {X 0,Y 324.555,Z 758.756,A -85,B 0,C 180,E1 -15092.061,E2 -15092.061} C_VEL
LIN {X 0,Y 325.992,Z 749.733,A -85,B 0,C 180,E1 -15093.599,E2 -15093.599} C_VEL
LIN {X 0,Y 327.49,Z 738.786,A -85,B 0,C 180,E1 -15095.092,E2 -15095.092} C_VEL
LIN {X 0,Y 328.736,Z 728.479,A -85,B 0,C 180,E1 -15096.215,E2 -15096.215} C_VEL
LIN {X 0,Y 329.874,Z 716.884,A -85,B 0,C 180,E1 -15097.211,E2 -15097.211} C_VEL
LIN {X 0,Y 330.728,Z 703.785,A -85,B 0,C 180,E1 -15098.046,E2 -15098.046} C_VEL
LIN {X 0,Y 331.268,Z 690.534,A -85,B 0,C 180,E1 -15098.626,E2 -15098.626} C_VEL
LIN {X 0,Y 333.567,Z 619.08,A -85,B 0,C 180,E1 -15100.402,E2 -15100.402} C_VEL
LIN {X 0,Y 326.035,Z 603.293,A -85,B 0,C 180,E1 -15101.63,E2 -15101.63} C_VEL
LIN {X 0,Y 321.019,Z 594.047,A -85,B 0,C 180,E1 -15102.46,E2 -15102.46} C_VEL
LIN {X 0,Y 319.724,Z 591.179,A -85,B 0,C 180,E1 -15102.696,E2 -15102.696} C_VEL
LIN {X 0,Y 319.64,Z 590.672,A -85,B 0,C 180,E1 -15102.733,E2 -15102.733} C_VEL
LIN {X 0,Y 319.726,Z 590.661,A -85,B 0,C 180,E1 -15106.007,E2 -15106.007} C_VEL
LIN {X 0,Y 319.752,Z 590.655,A -85,B 0,C 180,E1 -15109.873,E2 -15109.873} C_VEL
LIN {X 0,Y 319.927,Z 590.632,A -85,B 0,C 180,E1 -15112.426,E2 -15112.426} C_VEL
LIN {X 0,Y 319.744,Z 590.653,A -85,B 0,C 180,E1 -15114.956,E2 -15114.956} C_VEL
LIN {X 0,Y 319.985,Z 590.622,A -85,B 0,C 180,E1 -15117.482,E2 -15117.482} C_VEL
LIN {X 0,Y 320.161,Z 590.602,A -85,B 0,C 180,E1 -15120,E2 -15120} C_VEL
LIN {X 0,Y 319.985,Z 590.625,A -85,B 0,C 180,E1 -15122.518,E2 -15122.518} C_VEL
LIN {X 0,Y 319.942,Z 590.626,A -85,B 0,C 180,E1 -15126.306,E2 -15126.306} C_VEL
LIN {X 0,Y 319.835,Z 590.641,A -85,B 0,C 180,E1 -15128.848,E2 -15128.848} C_VEL
LIN {X 0,Y 319.678,Z 590.655,A -85,B 0,C 180,E1 -15132.7,E2 -15132.7} C_VEL
LIN {X 0,Y 319.692,Z 590.656,A -85,B 0,C 180,E1 -15135.296,E2 -15135.296} C_VEL
LIN {X 0,Y 319.669,Z 590.659,A -85,B 0,C 180,E1 -15139.255,E2 -15139.255} C_VEL
LIN {X 0,Y 319.564,Z 590.672,A -85,B 0,C 180,E1 -15143.32,E2 -15143.32} C_VEL
LIN {X 0,Y 319.629,Z 590.672,A -85,B 0,C 180,E1 -15146.089,E2 -15146.089} C_VEL
LIN {X 0,Y 319.584,Z 590.677,A -85,B 0,C 180,E1 -15148.934,E2 -15148.934} C_VEL
LIN {X 0,Y 319.528,Z 590.682,A -85,B 0,C 180,E1 -15151.862,E2 -15151.862} C_VEL
LIN {X 0,Y 319.575,Z 590.677,A -85,B 0,C 180,E1 -15155.544,E2 -15155.544} C_VEL
LIN {X 0,Y 319.595,Z 590.676,A -85,B 0,C 180,E1 -15158.005,E2 -15158.005} C_VEL
LIN {X 0,Y 319.592,Z 590.672,A -85,B 0,C 180,E1 -15161.612,E2 -15161.612} C_VEL
LIN {X 0,Y 319.572,Z 590.679,A -85,B 0,C 180,E1 -15165.274,E2 -15165.274} C_VEL
LIN {X 0,Y 319.545,Z 590.685,A -85,B 0,C 180,E1 -15168.716,E2 -15168.716} C_VEL
LIN {X 0,Y 319.58,Z 590.677,A -85,B 0,C 180,E1 -15172.344,E2 -15172.344} C_VEL
LIN {X 0,Y 319.606,Z 590.741,A -85,B 0,C 180,E1 -15172.892,E2 -15172.892} C_VEL
LIN {X 0,Y 322.17,Z 600.511,A -85,B 0,C 180,E1 -15175.992,E2 -15175.992} C_VEL
LIN {X 0,Y 324.585,Z 610.928,A -85,B 0,C 180,E1 -15179.024,E2 -15179.024} C_VEL
LIN {X 0,Y 326.108,Z 619.55,A -85,B 0,C 180,E1 -15181.347,E2 -15181.347} C_VEL
LIN {X 0,Y 324.685,Z 629.612,A -85,B 0,C 180,E1 -15183.698,E2 -15183.698} C_VEL
LIN {X 0,Y 329.092,Z 654.8,A -85,B 0,C 180,E1 -15184.869,E2 -15184.869} C_VEL
LIN {X 0,Y 332.077,Z 681.609,A -85,B 0,C 180,E1 -15185.89,E2 -15185.89} C_VEL
LIN {X 0,Y 330.179,Z 741.239,A -85,B 0,C 180,E1 -15187.375,E2 -15187.375} C_VEL
LIN {X 0,Y 329.108,Z 755.442,A -85,B 0,C 180,E1 -15187.974,E2 -15187.974} C_VEL
LIN {X 0,Y 327.761,Z 768.447,A -85,B 0,C 180,E1 -15188.787,E2 -15188.787} C_VEL
LIN {X 0,Y 326.13,Z 780.851,A -85,B 0,C 180,E1 -15189.831,E2 -15189.831} C_VEL
LIN {X 0,Y 324.588,Z 792.031,A -85,B 0,C 180,E1 -15191.048,E2 -15191.048} C_VEL
LIN {X 0,Y 322.817,Z 803.159,A -85,B 0,C 180,E1 -15192.582,E2 -15192.582} C_VEL
LIN {X 0,Y 321.436,Z 813.266,A -85,B 0,C 180,E1 -15194.334,E2 -15194.334} C_VEL
LIN {X 0,Y 320.116,Z 821.191,A -85,B 0,C 180,E1 -15196.025,E2 -15196.025} C_VEL
LIN {X 0,Y 319.167,Z 828.377,A -85,B 0,C 180,E1 -15197.926,E2 -15197.926} C_VEL
LIN {X 0,Y 318.516,Z 834.182,A -85,B 0,C 180,E1 -15199.833,E2 -15199.833} C_VEL
LIN {X 0,Y 318.21,Z 838.799,A -85,B 0,C 180,E1 -15201.746,E2 -15201.746} C_VEL
LIN {X 0,Y 318.123,Z 842.539,A -85,B 0,C 180,E1 -15203.798,E2 -15203.798} C_VEL
LIN {X 0,Y 318.104,Z 845.462,A -85,B 0,C 180,E1 -15206.2,E2 -15206.2} C_VEL
LIN {X 0,Y 318.303,Z 846.377,A -85,B 0,C 180,E1 -15207.469,E2 -15207.469} C_VEL
LIN {X 0,Y 318.349,Z 846.858,A -85,B 0,C 180,E1 -15208.735,E2 -15208.735} C_VEL
LIN {X 0,Y 318.44,Z 846.938,A -85,B 0,C 180,E1 -15210,E2 -15210} C_VEL
LIN {X 0,Y 318.383,Z 846.594,A -85,B 0,C 180,E1 -15211.265,E2 -15211.265} C_VEL
LIN {X 0,Y 318.35,Z 845.789,A -85,B 0,C 180,E1 -15212.531,E2 -15212.531} C_VEL
LIN {X 0,Y 318.131,Z 841.721,A -85,B 0,C 180,E1 -15216.214,E2 -15216.214} C_VEL
LIN {X 0,Y 318.189,Z 838.329,A -85,B 0,C 180,E1 -15218.254,E2 -15218.254} C_VEL
LIN {X 0,Y 318.52,Z 834.065,A -85,B 0,C 180,E1 -15220.167,E2 -15220.167} C_VEL
LIN {X 0,Y 319.369,Z 827.606,A -85,B 0,C 180,E1 -15222.389,E2 -15222.389} C_VEL
LIN {X 0,Y 320.376,Z 820.595,A -85,B 0,C 180,E1 -15224.287,E2 -15224.287} C_VEL
LIN {X 0,Y 321.652,Z 812.441,A -85,B 0,C 180,E1 -15226.056,E2 -15226.056} C_VEL
LIN {X 0,Y 323.26,Z 802.905,A -85,B 0,C 180,E1 -15227.72,E2 -15227.72} C_VEL
LIN {X 0,Y 324.888,Z 793.098,A -85,B 0,C 180,E1 -15229.097,E2 -15229.097} C_VEL
LIN {X 0,Y 326.504,Z 782.268,A -85,B 0,C 180,E1 -15230.309,E2 -15230.309} C_VEL
LIN {X 0,Y 328.146,Z 770.153,A -85,B 0,C 180,E1 -15231.351,E2 -15231.351} C_VEL
LIN {X 0,Y 329.559,Z 757.433,A -85,B 0,C 180,E1 -15232.159,E2 -15232.159} C_VEL
LIN {X 0,Y 330.55,Z 744.478,A -85,B 0,C 180,E1 -15232.714,E2 -15232.714} C_VEL
LIN {X 0,Y 331.089,Z 726.496,A -85,B 0,C 180,E1 -15233.173,E2 -15233.173} C_VEL
LIN {X 0,Y 332.191,Z 678.121,A -85,B 0,C 180,E1 -15234.241,E2 -15234.241} C_VEL
LIN {X 0,Y 329.176,Z 650.173,A -85,B 0,C 180,E1 -15235.201,E2 -15235.201} C_VEL
LIN {X 0,Y 325.09,Z 622.071,A -85,B 0,C 180,E1 -15236.306,E2 -15236.306} C_VEL
LIN {X 0,Y 325.611,Z 617.555,A -85,B 0,C 180,E1 -15237.181,E2 -15237.181} C_VEL
LIN {X 0,Y 323.27,Z 606.468,A -85,B 0,C 180,E1 -15239.586,E2 -15239.586} C_VEL
LIN {X 0,Y 319.562,Z 590.68,A -85,B 0,C 180,E1 -15243.198,E2 -15243.198} C_VEL
LIN {X 0,Y 319.559,Z 590.681,A -85,B 0,C 180,E1 -15246.426,E2 -15246.426} C_VEL
LIN {X 0,Y 319.562,Z 590.677,A -85,B 0,C 180,E1 -15249.669,E2 -15249.669} C_VEL
LIN {X 0,Y 319.586,Z 590.675,A -85,B 0,C 180,E1 -15253.473,E2 -15253.473} C_VEL
LIN {X 0,Y 319.6,Z 590.672,A -85,B 0,C 180,E1 -15257.024,E2 -15257.024} C_VEL
LIN {X 0,Y 319.581,Z 590.665,A -85,B 0,C 180,E1 -15260.376,E2 -15260.376} C_VEL
LIN {X 0,Y 319.556,Z 590.678,A -85,B 0,C 180,E1 -15263.572,E2 -15263.572} C_VEL
LIN {X 0,Y 319.573,Z 590.671,A -85,B 0,C 180,E1 -15266.685,E2 -15266.685} C_VEL
LIN {X 0,Y 319.588,Z 590.671,A -85,B 0,C 180,E1 -15269.616,E2 -15269.616} C_VEL
LIN {X 0,Y 319.603,Z 590.665,A -85,B 0,C 180,E1 -15272.498,E2 -15272.498} C_VEL
LIN {X 0,Y 319.598,Z 590.67,A -85,B 0,C 180,E1 -15275.303,E2 -15275.303} C_VEL
LIN {X 0,Y 319.59,Z 590.657,A -85,B 0,C 180,E1 -15278.047,E2 -15278.047} C_VEL
LIN {X 0,Y 319.682,Z 590.663,A -85,B 0,C 180,E1 -15280.962,E2 -15280.962} C_VEL
LIN {X 0,Y 319.724,Z 590.647,A -85,B 0,C 180,E1 -15285.276,E2 -15285.276} C_VEL
LIN {X 0,Y 319.745,Z 590.644,A -85,B 0,C 180,E1 -15289.872,E2 -15289.872} C_VEL
LIN {X 0,Y 319.906,Z 590.62,A -85,B 0,C 180,E1 -15292.426,E2 -15292.426} C_VEL
LIN {X 0,Y 319.743,Z 590.656,A -85,B 0,C 180,E1 -15294.956,E2 -15294.956} C_VEL
LIN {X 0,Y 319.985,Z 590.609,A -85,B 0,C 180,E1 -15297.482,E2 -15297.482} C_VEL
LIN {X 0,Y 320.144,Z 590.595,A -85,B 0,C 180,E1 -15300,E2 -15300} C_VEL
LIN {X 0,Y 320.001,Z 590.626,A -85,B 0,C 180,E1 -15302.518,E2 -15302.518} C_VEL
LIN {X 0,Y 319.92,Z 590.615,A -85,B 0,C 180,E1 -15306.605,E2 -15306.605} C_VEL
LIN {X 0,Y 319.835,Z 590.646,A -85,B 0,C 180,E1 -15308.848,E2 -15308.848} C_VEL
LIN {X 0,Y 319.673,Z 590.647,A -85,B 0,C 180,E1 -15312.7,E2 -15312.7} C_VEL
LIN {X 0,Y 319.692,Z 590.664,A -85,B 0,C 180,E1 -15315.296,E2 -15315.296} C_VEL
LIN {X 0,Y 319.667,Z 590.651,A -85,B 0,C 180,E1 -15319.256,E2 -15319.256} C_VEL
LIN {X 0,Y 319.562,Z 590.671,A -85,B 0,C 180,E1 -15323.32,E2 -15323.32} C_VEL
LIN {X 0,Y 319.629,Z 590.666,A -85,B 0,C 180,E1 -15326.089,E2 -15326.089} C_VEL
LIN {X 0,Y 319.584,Z 590.668,A -85,B 0,C 180,E1 -15328.934,E2 -15328.934} C_VEL
LIN {X 0,Y 319.533,Z 590.682,A -85,B 0,C 180,E1 -15331.862,E2 -15331.862} C_VEL
LIN {X 0,Y 319.575,Z 590.674,A -85,B 0,C 180,E1 -15335.544,E2 -15335.544} C_VEL
LIN {X 0,Y 319.578,Z 590.676,A -85,B 0,C 180,E1 -15338.008,E2 -15338.008} C_VEL
LIN {X 0,Y 319.564,Z 590.649,A -85,B 0,C 180,E1 -15341.606,E2 -15341.606} C_VEL
LIN {X 0,Y 319.516,Z 590.687,A -85,B 0,C 180,E1 -15345.264,E2 -15345.264} C_VEL
LIN {X 0,Y 319.525,Z 590.669,A -85,B 0,C 180,E1 -15348.713,E2 -15348.713} C_VEL
LIN {X 0,Y 319.575,Z 590.702,A -85,B 0,C 180,E1 -15351.285,E2 -15351.285} C_VEL
LIN {X 0,Y 320.519,Z 593.464,A -85,B 0,C 180,E1 -15351.459,E2 -15351.459} C_VEL
LIN {X 0,Y 325.286,Z 602.093,A -85,B 0,C 180,E1 -15352.182,E2 -15352.182} C_VEL
LIN {X 0,Y 331.381,Z 614.082,A -85,B 0,C 180,E1 -15353.088,E2 -15353.088} C_VEL
LIN {X 0,Y 334.171,Z 620.396,A -85,B 0,C 180,E1 -15353.508,E2 -15353.508} C_VEL
LIN {X 0,Y 332.495,Z 685.592,A -85,B 0,C 180,E1 -15354.928,E2 -15354.928} C_VEL
LIN {X 0,Y 332.056,Z 698.174,A -85,B 0,C 180,E1 -15355.375,E2 -15355.375} C_VEL
LIN {X 0,Y 331.323,Z 710.618,A -85,B 0,C 180,E1 -15356.055,E2 -15356.055} C_VEL
LIN {X 0,Y 330.205,Z 722.664,A -85,B 0,C 180,E1 -15356.949,E2 -15356.949} C_VEL
LIN {X 0,Y 328.881,Z 734.042,A -85,B 0,C 180,E1 -15358.07,E2 -15358.07} C_VEL
LIN {X 0,Y 327.26,Z 745.341,A -85,B 0,C 180,E1 -15359.484,E2 -15359.484} C_VEL
LIN {X 0,Y 325.753,Z 754.705,A -85,B 0,C 180,E1 -15360.96,E2 -15360.96} C_VEL
LIN {X 0,Y 324.215,Z 763.622,A -85,B 0,C 180,E1 -15362.718,E2 -15362.718} C_VEL
LIN {X 0,Y 322.758,Z 771.054,A -85,B 0,C 180,E1 -15364.53,E2 -15364.53} C_VEL
LIN {X 0,Y 321.641,Z 776.655,A -85,B 0,C 180,E1 -15366.226,E2 -15366.226} C_VEL
LIN {X 0,Y 320.618,Z 781.664,A -85,B 0,C 180,E1 -15368.122,E2 -15368.122} C_VEL
LIN {X 0,Y 319.812,Z 785.62,A -85,B 0,C 180,E1 -15370.086,E2 -15370.086} C_VEL
LIN {X 0,Y 319.171,Z 788.476,A -85,B 0,C 180,E1 -15372.045,E2 -15372.045} C_VEL
LIN {X 0,Y 318.824,Z 789.797,A -85,B 0,C 180,E1 -15373.348,E2 -15373.348} C_VEL
LIN {X 0,Y 318.596,Z 790.712,A -85,B 0,C 180,E1 -15374.651,E2 -15374.651} C_VEL
LIN {X 0,Y 318.416,Z 791.259,A -85,B 0,C 180,E1 -15376.206,E2 -15376.206} C_VEL
LIN {X 0,Y 318.27,Z 790.965,A -85,B 0,C 180,E1 -15378.537,E2 -15378.537} C_VEL
LIN {X 0,Y 318.296,Z 790.251,A -85,B 0,C 180,E1 -15379.826,E2 -15379.826} C_VEL
LIN {X 0,Y 318.404,Z 789.108,A -85,B 0,C 180,E1 -15381.112,E2 -15381.112} C_VEL
LIN {X 0,Y 318.676,Z 786.76,A -85,B 0,C 180,E1 -15382.941,E2 -15382.941} C_VEL
LIN {X 0,Y 319.041,Z 783.12,A -85,B 0,C 180,E1 -15384.945,E2 -15384.945} C_VEL
LIN {X 0,Y 319.499,Z 778.542,A -85,B 0,C 180,E1 -15386.848,E2 -15386.848} C_VEL
LIN {X 0,Y 320.305,Z 771.644,A -85,B 0,C 180,E1 -15389.057,E2 -15389.057} C_VEL
LIN {X 0,Y 321.154,Z 764.155,A -85,B 0,C 180,E1 -15390.94,E2 -15390.94} C_VEL
LIN {X 0,Y 322.354,Z 754.735,A -85,B 0,C 180,E1 -15392.812,E2 -15392.812} C_VEL
LIN {X 0,Y 323.442,Z 745.048,A -85,B 0,C 180,E1 -15394.361,E2 -15394.361} C_VEL
LIN {X 0,Y 324.538,Z 734.143,A -85,B 0,C 180,E1 -15395.748,E2 -15395.748} C_VEL
LIN {X 0,Y 325.613,Z 722.838,A -85,B 0,C 180,E1 -15396.88,E2 -15396.88} C_VEL
LIN {X 0,Y 326.451,Z 710.727,A -85,B 0,C 180,E1 -15397.81,E2 -15397.81} C_VEL
LIN {X 0,Y 327.027,Z 697.651,A -85,B 0,C 180,E1 -15398.535,E2 -15398.535} C_VEL
LIN {X 0,Y 327.415,Z 684.458,A -85,B 0,C 180,E1 -15399,E2 -15399} C_VEL
LIN {X 0,Y 328.791,Z 614.241,A -85,B 0,C 180,E1 -15400.522,E2 -15400.522} C_VEL
LIN {X 0,Y 320.541,Z 593.185,A -85,B 0,C 180,E1 -15401.532,E2 -15401.532} C_VEL
LIN {X 0,Y 319.731,Z 590.658,A -85,B 0,C 180,E1 -15401.651,E2 -15401.651} C_VEL
LIN {X 0,Y 319.701,Z 590.659,A -85,B 0,C 180,E1 -15405.295,E2 -15405.295} C_VEL
LIN {X 0,Y 319.674,Z 590.664,A -85,B 0,C 180,E1 -15409.254,E2 -15409.254} C_VEL
LIN {X 0,Y 319.6,Z 590.675,A -85,B 0,C 180,E1 -15411.909,E2 -15411.909} C_VEL
LIN {X 0,Y 321.687,Z 596.174,A -85,B 0,C 180,E1 -15412.2,E2 -15412.2} C_VEL
LIN {X 0,Y 329.507,Z 615.548,A -85,B 0,C 180,E1 -15413.219,E2 -15413.219} C_VEL
LIN {X 0,Y 327.898,Z 677.867,A -85,B 0,C 180,E1 -15414.688,E2 -15414.688} C_VEL
LIN {X 0,Y 327.061,Z 683.689,A -85,B 0,C 180,E1 -15414.791,E2 -15414.791} C_VEL
LIN {X 0,Y 324.044,Z 693.102,A -85,B 0,C 180,E1 -15414.94,E2 -15414.94} C_VEL
LIN {X 0,Y 321.076,Z 702.431,A -85,B 0,C 180,E1 -15415.229,E2 -15415.229} C_VEL
LIN {X 0,Y 320.224,Z 707.973,A -85,B 0,C 180,E1 -15415.524,E2 -15415.524} C_VEL
LIN {X 0,Y 319.322,Z 719.764,A -85,B 0,C 180,E1 -15416.378,E2 -15416.378} C_VEL
LIN {X 0,Y 318.361,Z 730.906,A -85,B 0,C 180,E1 -15417.44,E2 -15417.44} C_VEL
LIN {X 0,Y 317.148,Z 742.518,A -85,B 0,C 180,E1 -15418.843,E2 -15418.843} C_VEL
LIN {X 0,Y 316.038,Z 752.302,A -85,B 0,C 180,E1 -15420.317,E2 -15420.317} C_VEL
LIN {X 0,Y 314.949,Z 761.356,A -85,B 0,C 180,E1 -15422.009,E2 -15422.009} C_VEL
LIN {X 0,Y 313.783,Z 770.133,A -85,B 0,C 180,E1 -15424.051,E2 -15424.051} C_VEL
LIN {X 0,Y 312.968,Z 776.95,A -85,B 0,C 180,E1 -15426.058,E2 -15426.058} C_VEL
LIN {X 0,Y 312.298,Z 782.223,A -85,B 0,C 180,E1 -15428.034,E2 -15428.034} C_VEL
LIN {X 0,Y 311.811,Z 786.229,A -85,B 0,C 180,E1 -15429.974,E2 -15429.974} C_VEL
LIN {X 0,Y 311.438,Z 789.138,A -85,B 0,C 180,E1 -15431.867,E2 -15431.867} C_VEL
LIN {X 0,Y 311.163,Z 791.599,A -85,B 0,C 180,E1 -15434.44,E2 -15434.44} C_VEL
LIN {X 0,Y 311.156,Z 792.372,A -85,B 0,C 180,E1 -15436.283,E2 -15436.283} C_VEL
LIN {X 0,Y 311.324,Z 792.329,A -85,B 0,C 180,E1 -15438.154,E2 -15438.154} C_VEL
LIN {X 0,Y 311.608,Z 791.42,A -85,B 0,C 180,E1 -15440.069,E2 -15440.069} C_VEL
LIN {X 0,Y 312.268,Z 788.827,A -85,B 0,C 180,E1 -15442.579,E2 -15442.579} C_VEL
LIN {X 0,Y 312.797,Z 786.194,A -85,B 0,C 180,E1 -15444.255,E2 -15444.255} C_VEL
LIN {X 0,Y 313.536,Z 782.537,A -85,B 0,C 180,E1 -15446.031,E2 -15446.031} C_VEL
LIN {X 0,Y 314.632,Z 777.043,A -85,B 0,C 180,E1 -15448.081,E2 -15448.081} C_VEL
LIN {X 0,Y 316.003,Z 769.926,A -85,B 0,C 180,E1 -15450.152,E2 -15450.152} C_VEL
LIN {X 0,Y 317.404,Z 762.233,A -85,B 0,C 180,E1 -15451.933,E2 -15451.933} C_VEL
LIN {X 0,Y 319.033,Z 752.739,A -85,B 0,C 180,E1 -15453.683,E2 -15453.683} C_VEL
LIN {X 0,Y 320.665,Z 742.215,A -85,B 0,C 180,E1 -15455.236,E2 -15455.236} C_VEL
LIN {X 0,Y 321.985,Z 731.893,A -85,B 0,C 180,E1 -15456.45,E2 -15456.45} C_VEL
LIN {X 0,Y 323.229,Z 719.981,A -85,B 0,C 180,E1 -15457.551,E2 -15457.551} C_VEL
LIN {X 0,Y 324.272,Z 707.084,A -85,B 0,C 180,E1 -15458.446,E2 -15458.446} C_VEL
LIN {X 0,Y 324.888,Z 694.196,A -85,B 0,C 180,E1 -15459.068,E2 -15459.068} C_VEL
LIN {X 0,Y 325.501,Z 674.149,A -85,B 0,C 180,E1 -15459.636,E2 -15459.636} C_VEL
LIN {X 0,Y 327.306,Z 620.98,A -85,B 0,C 180,E1 -15460.976,E2 -15460.976} C_VEL
LIN {X 0,Y 319.368,Z 604.545,A -85,B 0,C 180,E1 -15462.329,E2 -15462.329} C_VEL
LIN {X 0,Y 314.065,Z 595.042,A -85,B 0,C 180,E1 -15463.255,E2 -15463.255} C_VEL
LIN {X 0,Y 312.716,Z 592.079,A -85,B 0,C 180,E1 -15463.517,E2 -15463.517} C_VEL
LIN {X 0,Y 312.626,Z 591.544,A -85,B 0,C 180,E1 -15463.596,E2 -15463.596} C_VEL
LIN {X 0,Y 312.63,Z 591.544,A -85,B 0,C 180,E1 -15467.009,E2 -15467.009} C_VEL
LIN {X 0,Y 312.827,Z 591.519,A -85,B 0,C 180,E1 -15471.296,E2 -15471.296} C_VEL
LIN {X 0,Y 312.905,Z 591.509,A -85,B 0,C 180,E1 -15473.552,E2 -15473.552} C_VEL
LIN {X 0,Y 312.932,Z 591.5,A -85,B 0,C 180,E1 -15477.426,E2 -15477.426} C_VEL
LIN {X 0,Y 313.113,Z 591.48,A -85,B 0,C 180,E1 -15480,E2 -15480} C_VEL
LIN {X 0,Y 312.931,Z 591.503,A -85,B 0,C 180,E1 -15482.574,E2 -15482.574} C_VEL
LIN {X 0,Y 312.9,Z 591.502,A -85,B 0,C 180,E1 -15486.448,E2 -15486.448} C_VEL
LIN {X 0,Y 312.781,Z 591.518,A -85,B 0,C 180,E1 -15489.049,E2 -15489.049} C_VEL
LIN {X 0,Y 312.629,Z 591.53,A -85,B 0,C 180,E1 -15492.991,E2 -15492.991} C_VEL
LIN {X 0,Y 312.631,Z 591.535,A -85,B 0,C 180,E1 -15495.65,E2 -15495.65} C_VEL
LIN {X 0,Y 312.625,Z 591.537,A -85,B 0,C 180,E1 -15499.237,E2 -15499.237} C_VEL
LIN {X 0,Y 312.539,Z 591.55,A -85,B 0,C 180,E1 -15502.79,E2 -15502.79} C_VEL
LIN {X 0,Y 312.597,Z 591.547,A -85,B 0,C 180,E1 -15505.936,E2 -15505.936} C_VEL
LIN {X 0,Y 312.54,Z 591.553,A -85,B 0,C 180,E1 -15509.651,E2 -15509.651} C_VEL
LIN {X 0,Y 312.515,Z 591.551,A -85,B 0,C 180,E1 -15513.69,E2 -15513.69} C_VEL
LIN {X 0,Y 312.548,Z 591.552,A -85,B 0,C 180,E1 -15517.382,E2 -15517.382} C_VEL
LIN {X 0,Y 312.522,Z 591.556,A -85,B 0,C 180,E1 -15520.704,E2 -15520.704} C_VEL
LIN {X 0,Y 312.529,Z 591.554,A -85,B 0,C 180,E1 -15524.196,E2 -15524.196} C_VEL
LIN {X 0,Y 312.531,Z 591.556,A -85,B 0,C 180,E1 -15527.909,E2 -15527.909} C_VEL
LIN {X 0,Y 312.577,Z 591.715,A -85,B 0,C 180,E1 -15532.157,E2 -15532.157} C_VEL
LIN {X 0,Y 315.328,Z 602.031,A -85,B 0,C 180,E1 -15535.553,E2 -15535.553} C_VEL
LIN {X 0,Y 317.416,Z 611.009,A -85,B 0,C 180,E1 -15538.275,E2 -15538.275} C_VEL
LIN {X 0,Y 319.027,Z 619.405,A -85,B 0,C 180,E1 -15540.65,E2 -15540.65} C_VEL
LIN {X 0,Y 319.145,Z 622.854,A -85,B 0,C 180,E1 -15541.54,E2 -15541.54} C_VEL
LIN {X 0,Y 318.185,Z 628.933,A -85,B 0,C 180,E1 -15542.974,E2 -15542.974} C_VEL
LIN {X 0,Y 322.558,Z 653.709,A -85,B 0,C 180,E1 -15544.183,E2 -15544.183} C_VEL
LIN {X 0,Y 325.442,Z 678.563,A -85,B 0,C 180,E1 -15545.186,E2 -15545.186} C_VEL
LIN {X 0,Y 325.767,Z 682.849,A -85,B 0,C 180,E1 -15545.338,E2 -15545.338} C_VEL
LIN {X 0,Y 323.865,Z 740.336,A -85,B 0,C 180,E1 -15546.798,E2 -15546.798} C_VEL
LIN {X 0,Y 322.787,Z 754.302,A -85,B 0,C 180,E1 -15547.392,E2 -15547.392} C_VEL
LIN {X 0,Y 321.434,Z 766.925,A -85,B 0,C 180,E1 -15548.18,E2 -15548.18} C_VEL
LIN {X 0,Y 319.7,Z 779.455,A -85,B 0,C 180,E1 -15549.239,E2 -15549.239} C_VEL
LIN {X 0,Y 318.081,Z 790.734,A -85,B 0,C 180,E1 -15550.477,E2 -15550.477} C_VEL
LIN {X 0,Y 316.367,Z 800.981,A -85,B 0,C 180,E1 -15551.881,E2 -15551.881} C_VEL
LIN {X 0,Y 314.996,Z 809.926,A -85,B 0,C 180,E1 -15553.393,E2 -15553.393} C_VEL
LIN {X 0,Y 313.75,Z 818.097,A -85,B 0,C 180,E1 -15555.073,E2 -15555.073} C_VEL
LIN {X 0,Y 312.513,Z 825.771,A -85,B 0,C 180,E1 -15557.004,E2 -15557.004} C_VEL
LIN {X 0,Y 311.658,Z 831.977,A -85,B 0,C 180,E1 -15558.95,E2 -15558.95} C_VEL
LIN {X 0,Y 311.225,Z 836.929,A -85,B 0,C 180,E1 -15560.905,E2 -15560.905} C_VEL
LIN {X 0,Y 311.024,Z 840.756,A -85,B 0,C 180,E1 -15562.861,E2 -15562.861} C_VEL
LIN {X 0,Y 311.022,Z 843.55,A -85,B 0,C 180,E1 -15564.814,E2 -15564.814} C_VEL
LIN {X 0,Y 311.024,Z 844.887,A -85,B 0,C 180,E1 -15566.113,E2 -15566.113} C_VEL
LIN {X 0,Y 311.219,Z 845.775,A -85,B 0,C 180,E1 -15567.411,E2 -15567.411} C_VEL
LIN {X 0,Y 311.285,Z 846.242,A -85,B 0,C 180,E1 -15568.706,E2 -15568.706} C_VEL
LIN {X 0,Y 311.369,Z 846.305,A -85,B 0,C 180,E1 -15570,E2 -15570} C_VEL
LIN {X 0,Y 311.318,Z 845.934,A -85,B 0,C 180,E1 -15571.294,E2 -15571.294} C_VEL
LIN {X 0,Y 311.285,Z 845.1,A -85,B 0,C 180,E1 -15572.588,E2 -15572.588} C_VEL
LIN {X 0,Y 311.047,Z 841.448,A -85,B 0,C 180,E1 -15576.191,E2 -15576.191} C_VEL
LIN {X 0,Y 311.125,Z 837.878,A -85,B 0,C 180,E1 -15578.443,E2 -15578.443} C_VEL
LIN {X 0,Y 311.493,Z 833.664,A -85,B 0,C 180,E1 -15580.399,E2 -15580.399} C_VEL
LIN {X 0,Y 312.402,Z 827.258,A -85,B 0,C 180,E1 -15582.67,E2 -15582.67} C_VEL
LIN {X 0,Y 313.478,Z 820.315,A -85,B 0,C 180,E1 -15584.608,E2 -15584.608} C_VEL
LIN {X 0,Y 314.731,Z 812.593,A -85,B 0,C 180,E1 -15586.349,E2 -15586.349} C_VEL
LIN {X 0,Y 316.475,Z 802.811,A -85,B 0,C 180,E1 -15588.113,E2 -15588.113} C_VEL
LIN {X 0,Y 318.2,Z 793.116,A -85,B 0,C 180,E1 -15589.515,E2 -15589.515} C_VEL
LIN {X 0,Y 319.861,Z 782.504,A -85,B 0,C 180,E1 -15590.75,E2 -15590.75} C_VEL
LIN {X 0,Y 321.554,Z 770.624,A -85,B 0,C 180,E1 -15591.811,E2 -15591.811} C_VEL
LIN {X 0,Y 323.01,Z 758.288,A -85,B 0,C 180,E1 -15592.633,E2 -15592.633} C_VEL
LIN {X 0,Y 324.078,Z 746.061,A -85,B 0,C 180,E1 -15593.204,E2 -15593.204} C_VEL
LIN {X 0,Y 324.639,Z 731.577,A -85,B 0,C 180,E1 -15593.618,E2 -15593.618} C_VEL
LIN {X 0,Y 325.911,Z 678.914,A -85,B 0,C 180,E1 -15594.801,E2 -15594.801} C_VEL
LIN {X 0,Y 322.95,Z 651.067,A -85,B 0,C 180,E1 -15595.783,E2 -15595.783} C_VEL
LIN {X 0,Y 318.494,Z 620.333,A -85,B 0,C 180,E1 -15597.046,E2 -15597.046} C_VEL
LIN {X 0,Y 318.523,Z 617.613,A -85,B 0,C 180,E1 -15597.603,E2 -15597.603} C_VEL
LIN {X 0,Y 315.268,Z 603.192,A -85,B 0,C 180,E1 -15600.844,E2 -15600.844} C_VEL
LIN {X 0,Y 312.539,Z 591.556,A -85,B 0,C 180,E1 -15603.629,E2 -15603.629} C_VEL
LIN {X 0,Y 312.54,Z 591.553,A -85,B 0,C 180,E1 -15607.382,E2 -15607.382} C_VEL
LIN {X 0,Y 312.499,Z 591.556,A -85,B 0,C 180,E1 -15610.706,E2 -15610.706} C_VEL
LIN {X 0,Y 312.527,Z 591.555,A -85,B 0,C 180,E1 -15614.195,E2 -15614.195} C_VEL
LIN {X 0,Y 312.545,Z 591.554,A -85,B 0,C 180,E1 -15617.905,E2 -15617.905} C_VEL
LIN {X 0,Y 312.554,Z 591.548,A -85,B 0,C 180,E1 -15621.904,E2 -15621.904} C_VEL
LIN {X 0,Y 312.502,Z 591.542,A -85,B 0,C 180,E1 -15625.789,E2 -15625.789} C_VEL
LIN {X 0,Y 312.523,Z 591.552,A -85,B 0,C 180,E1 -15628.854,E2 -15628.854} C_VEL
LIN {X 0,Y 312.569,Z 591.534,A -85,B 0,C 180,E1 -15631.824,E2 -15631.824} C_VEL
LIN {X 0,Y 312.579,Z 591.547,A -85,B 0,C 180,E1 -15634.71,E2 -15634.71} C_VEL
LIN {X 0,Y 312.581,Z 591.527,A -85,B 0,C 180,E1 -15637.528,E2 -15637.528} C_VEL
LIN {X 0,Y 312.631,Z 591.539,A -85,B 0,C 180,E1 -15641.656,E2 -15641.656} C_VEL
LIN {X 0,Y 312.687,Z 591.526,A -85,B 0,C 180,E1 -15645.686,E2 -15645.686} C_VEL
LIN {X 0,Y 312.691,Z 591.525,A -85,B 0,C 180,E1 -15649.641,E2 -15649.641} C_VEL
LIN {X 0,Y 312.847,Z 591.498,A -85,B 0,C 180,E1 -15652.254,E2 -15652.254} C_VEL
LIN {X 0,Y 312.713,Z 591.533,A -85,B 0,C 180,E1 -15654.842,E2 -15654.842} C_VEL
LIN {X 0,Y 312.985,Z 591.476,A -85,B 0,C 180,E1 -15658.713,E2 -15658.713} C_VEL
LIN {X 0,Y 312.987,Z 591.497,A -85,B 0,C 180,E1 -15661.287,E2 -15661.287} C_VEL
LIN {X 0,Y 312.69,Z 591.528,A -85,B 0,C 180,E1 -15663.866,E2 -15663.866} C_VEL
LIN {X 0,Y 312.885,Z 591.491,A -85,B 0,C 180,E1 -15666.587,E2 -15666.587} C_VEL
LIN {X 0,Y 312.78,Z 591.525,A -85,B 0,C 180,E1 -15669.049,E2 -15669.049} C_VEL
LIN {X 0,Y 312.626,Z 591.525,A -85,B 0,C 180,E1 -15672.991,E2 -15672.991} C_VEL
LIN {X 0,Y 312.631,Z 591.541,A -85,B 0,C 180,E1 -15675.65,E2 -15675.65} C_VEL
LIN {X 0,Y 312.623,Z 591.528,A -85,B 0,C 180,E1 -15679.236,E2 -15679.236} C_VEL
LIN {X 0,Y 312.539,Z 591.552,A -85,B 0,C 180,E1 -15682.789,E2 -15682.789} C_VEL
LIN {X 0,Y 312.597,Z 591.542,A -85,B 0,C 180,E1 -15685.936,E2 -15685.936} C_VEL
LIN {X 0,Y 312.541,Z 591.54,A -85,B 0,C 180,E1 -15689.65,E2 -15689.65} C_VEL
LIN {X 0,Y 312.515,Z 591.548,A -85,B 0,C 180,E1 -15693.69,E2 -15693.69} C_VEL
LIN {X 0,Y 312.536,Z 591.553,A -85,B 0,C 180,E1 -15697.384,E2 -15697.384} C_VEL
LIN {X 0,Y 312.496,Z 591.539,A -85,B 0,C 180,E1 -15700.708,E2 -15700.708} C_VEL
LIN {X 0,Y 312.51,Z 591.549,A -85,B 0,C 180,E1 -15704.199,E2 -15704.199} C_VEL
LIN {X 0,Y 312.483,Z 591.54,A -85,B 0,C 180,E1 -15707.919,E2 -15707.919} C_VEL
LIN {X 0,Y 312.525,Z 591.701,A -85,B 0,C 180,E1 -15710.524,E2 -15710.524} C_VEL
LIN {X 0,Y 313.692,Z 594.676,A -85,B 0,C 180,E1 -15710.736,E2 -15710.736} C_VEL
LIN {X 0,Y 318.223,Z 602.7,A -85,B 0,C 180,E1 -15711.45,E2 -15711.45} C_VEL
LIN {X 0,Y 325.752,Z 617.456,A -85,B 0,C 180,E1 -15712.615,E2 -15712.615} C_VEL
LIN {X 0,Y 327.9,Z 622.043,A -85,B 0,C 180,E1 -15712.945,E2 -15712.945} C_VEL
LIN {X 0,Y 326.22,Z 685.046,A -85,B 0,C 180,E1 -15714.34,E2 -15714.34} C_VEL
LIN {X 0,Y 325.751,Z 698.274,A -85,B 0,C 180,E1 -15714.797,E2 -15714.797} C_VEL
LIN {X 0,Y 324.995,Z 710.958,A -85,B 0,C 180,E1 -15715.498,E2 -15715.498} C_VEL
LIN {X 0,Y 323.834,Z 722.981,A -85,B 0,C 180,E1 -15716.399,E2 -15716.399} C_VEL
LIN {X 0,Y 322.455,Z 734.437,A -85,B 0,C 180,E1 -15717.541,E2 -15717.541} C_VEL
LIN {X 0,Y 320.802,Z 745.552,A -85,B 0,C 180,E1 -15718.95,E2 -15718.95} C_VEL
LIN {X 0,Y 319.319,Z 754.241,A -85,B 0,C 180,E1 -15720.317,E2 -15720.317} C_VEL
LIN {X 0,Y 317.791,Z 762.915,A -85,B 0,C 180,E1 -15722.006,E2 -15722.006} C_VEL
LIN {X 0,Y 316.13,Z 770.959,A -85,B 0,C 180,E1 -15723.956,E2 -15723.956} C_VEL
LIN {X 0,Y 314.981,Z 776.486,A -85,B 0,C 180,E1 -15725.621,E2 -15725.621} C_VEL
LIN {X 0,Y 313.813,Z 781.812,A -85,B 0,C 180,E1 -15727.622,E2 -15727.622} C_VEL
LIN {X 0,Y 312.95,Z 785.884,A -85,B 0,C 180,E1 -15729.63,E2 -15729.63} C_VEL
LIN {X 0,Y 312.241,Z 788.844,A -85,B 0,C 180,E1 -15731.633,E2 -15731.633} C_VEL
LIN {X 0,Y 311.845,Z 790.248,A -85,B 0,C 180,E1 -15732.964,E2 -15732.964} C_VEL
LIN {X 0,Y 311.418,Z 791.772,A -85,B 0,C 180,E1 -15735.627,E2 -15735.627} C_VEL
LIN {X 0,Y 311.283,Z 791.926,A -85,B 0,C 180,E1 -15736.952,E2 -15736.952} C_VEL
LIN {X 0,Y 311.225,Z 790.973,A -85,B 0,C 180,E1 -15739.592,E2 -15739.592} C_VEL
LIN {X 0,Y 311.307,Z 789.914,A -85,B 0,C 180,E1 -15740.908,E2 -15740.908} C_VEL
LIN {X 0,Y 311.606,Z 787.43,A -85,B 0,C 180,E1 -15742.925,E2 -15742.925} C_VEL
LIN {X 0,Y 311.922,Z 784.117,A -85,B 0,C 180,E1 -15744.829,E2 -15744.829} C_VEL
LIN {X 0,Y 312.429,Z 779.65,A -85,B 0,C 180,E1 -15746.776,E2 -15746.776} C_VEL
LIN {X 0,Y 313.227,Z 772.873,A -85,B 0,C 180,E1 -15749.036,E2 -15749.036} C_VEL
LIN {X 0,Y 314.088,Z 765.55,A -85,B 0,C 180,E1 -15750.962,E2 -15750.962} C_VEL
LIN {X 0,Y 315.102,Z 758.037,A -85,B 0,C 180,E1 -15752.557,E2 -15752.557} C_VEL
LIN {X 0,Y 316.289,Z 747.875,A -85,B 0,C 180,E1 -15754.301,E2 -15754.301} C_VEL
LIN {X 0,Y 317.385,Z 737.593,A -85,B 0,C 180,E1 -15755.719,E2 -15755.719} C_VEL
LIN {X 0,Y 318.442,Z 727.196,A -85,B 0,C 180,E1 -15756.86,E2 -15756.86} C_VEL
LIN {X 0,Y 319.438,Z 714.901,A -85,B 0,C 180,E1 -15757.903,E2 -15757.903} C_VEL
LIN {X 0,Y 320.102,Z 701.944,A -85,B 0,C 180,E1 -15758.721,E2 -15758.721} C_VEL
LIN {X 0,Y 320.564,Z 688.69,A -85,B 0,C 180,E1 -15759.265,E2 -15759.265} C_VEL
LIN {X 0,Y 321.972,Z 615.324,A -85,B 0,C 180,E1 -15760.92,E2 -15760.92} C_VEL
LIN {X 0,Y 313.349,Z 593.768,A -85,B 0,C 180,E1 -15762,E2 -15762} C_VEL
LIN {X 0,Y 312.695,Z 591.537,A -85,B 0,C 180,E1 -15762.102,E2 -15762.102} C_VEL
LIN {X 0,Y 312.64,Z 591.538,A -85,B 0,C 180,E1 -15765.649,E2 -15765.649} C_VEL
LIN {X 0,Y 312.653,Z 591.539,A -85,B 0,C 180,E1 -15769.248,E2 -15769.248} C_VEL
LIN {X 0,Y 312.553,Z 591.549,A -85,B 0,C 180,E1 -15771.431,E2 -15771.431} C_VEL
LIN {X 0,Y 314.373,Z 596.455,A -85,B 0,C 180,E1 -15771.71,E2 -15771.71} C_VEL
LIN {X 0,Y 322.779,Z 617.106,A -85,B 0,C 180,E1 -15772.821,E2 -15772.821} C_VEL
LIN {X 0,Y 320.965,Z 688.529,A -85,B 0,C 180,E1 -15774.584,E2 -15774.584} C_VEL
LIN {X 0,Y 320.506,Z 702.131,A -85,B 0,C 180,E1 -15775.181,E2 -15775.181} C_VEL
LIN {X 0,Y 320.224,Z 707.973,A -85,B 0,C 180,E1 -15775.524,E2 -15775.524} C_VEL
LIN {X 0,Y 319.228,Z 713.521,A -85,B 0,C 180,E1 -15775.851,E2 -15775.851} C_VEL
LIN {X 0,Y 315.727,Z 722.355,A -85,B 0,C 180,E1 -15776.384,E2 -15776.384} C_VEL
LIN {X 0,Y 312.171,Z 730.826,A -85,B 0,C 180,E1 -15777.061,E2 -15777.061} C_VEL
LIN {X 0,Y 311.098,Z 735.797,A -85,B 0,C 180,E1 -15777.609,E2 -15777.609} C_VEL
LIN {X 0,Y 309.951,Z 746.148,A -85,B 0,C 180,E1 -15778.99,E2 -15778.99} C_VEL
LIN {X 0,Y 308.696,Z 756.341,A -85,B 0,C 180,E1 -15780.675,E2 -15780.675} C_VEL
LIN {X 0,Y 307.674,Z 764.376,A -85,B 0,C 180,E1 -15782.31,E2 -15782.31} C_VEL
LIN {X 0,Y 306.517,Z 772.525,A -85,B 0,C 180,E1 -15784.368,E2 -15784.368} C_VEL
LIN {X 0,Y 305.76,Z 779.007,A -85,B 0,C 180,E1 -15786.439,E2 -15786.439} C_VEL
LIN {X 0,Y 305.129,Z 783.968,A -85,B 0,C 180,E1 -15788.453,E2 -15788.453} C_VEL
LIN {X 0,Y 304.629,Z 787.674,A -85,B 0,C 180,E1 -15790.418,E2 -15790.418} C_VEL
LIN {X 0,Y 304.282,Z 790.324,A -85,B 0,C 180,E1 -15792.345,E2 -15792.345} C_VEL
LIN {X 0,Y 304.095,Z 792.054,A -85,B 0,C 180,E1 -15794.238,E2 -15794.238} C_VEL
LIN {X 0,Y 304.077,Z 792.951,A -85,B 0,C 180,E1 -15796.102,E2 -15796.102} C_VEL
LIN {X 0,Y 304.227,Z 793.059,A -85,B 0,C 180,E1 -15797.938,E2 -15797.938} C_VEL
LIN {X 0,Y 304.504,Z 792.372,A -85,B 0,C 180,E1 -15799.741,E2 -15799.741} C_VEL
LIN {X 0,Y 305.165,Z 789.965,A -85,B 0,C 180,E1 -15802.429,E2 -15802.429} C_VEL
LIN {X 0,Y 306.025,Z 786.068,A -85,B 0,C 180,E1 -15804.961,E2 -15804.961} C_VEL
LIN {X 0,Y 307.097,Z 780.967,A -85,B 0,C 180,E1 -15807.272,E2 -15807.272} C_VEL
LIN {X 0,Y 308.526,Z 774.224,A -85,B 0,C 180,E1 -15809.547,E2 -15809.547} C_VEL
LIN {X 0,Y 310.082,Z 766.499,A -85,B 0,C 180,E1 -15811.578,E2 -15811.578} C_VEL
LIN {X 0,Y 311.745,Z 757.439,A -85,B 0,C 180,E1 -15813.453,E2 -15813.453} C_VEL
LIN {X 0,Y 313.325,Z 748.428,A -85,B 0,C 180,E1 -15814.952,E2 -15814.952} C_VEL
LIN {X 0,Y 314.761,Z 738.522,A -85,B 0,C 180,E1 -15816.303,E2 -15816.303} C_VEL
LIN {X 0,Y 316.186,Z 727.022,A -85,B 0,C 180,E1 -15817.54,E2 -15817.54} C_VEL
LIN {X 0,Y 317.522,Z 714.049,A -85,B 0,C 180,E1 -15818.605,E2 -15818.605} C_VEL
LIN {X 0,Y 318.358,Z 700.951,A -85,B 0,C 180,E1 -15819.386,E2 -15819.386} C_VEL
LIN {X 0,Y 318.888,Z 688.115,A -85,B 0,C 180,E1 -15819.884,E2 -15819.884} C_VEL
LIN {X 0,Y 321.185,Z 623.23,A -85,B 0,C 180,E1 -15821.563,E2 -15821.563} C_VEL
LIN {X 0,Y 314.25,Z 608.682,A -85,B 0,C 180,E1 -15822.801,E2 -15822.801} C_VEL
LIN {X 0,Y 307.155,Z 596.07,A -85,B 0,C 180,E1 -15824.097,E2 -15824.097} C_VEL
LIN {X 0,Y 305.812,Z 593.447,A -85,B 0,C 180,E1 -15824.364,E2 -15824.364} C_VEL
LIN {X 0,Y 305.59,Z 592.421,A -85,B 0,C 180,E1 -15824.465,E2 -15824.465} C_VEL
LIN {X 0,Y 305.599,Z 592.418,A -85,B 0,C 180,E1 -15828.055,E2 -15828.055} C_VEL
LIN {X 0,Y 305.806,Z 592.392,A -85,B 0,C 180,E1 -15832.074,E2 -15832.074} C_VEL
LIN {X 0,Y 305.685,Z 592.405,A -85,B 0,C 180,E1 -15834.723,E2 -15834.723} C_VEL
LIN {X 0,Y 305.952,Z 592.375,A -85,B 0,C 180,E1 -15838.684,E2 -15838.684} C_VEL
LIN {X 0,Y 305.951,Z 592.373,A -85,B 0,C 180,E1 -15841.316,E2 -15841.316} C_VEL
LIN {X 0,Y 305.842,Z 592.38,A -85,B 0,C 180,E1 -15846.598,E2 -15846.598} C_VEL
LIN {X 0,Y 305.729,Z 592.395,A -85,B 0,C 180,E1 -15849.26,E2 -15849.26} C_VEL
LIN {X 0,Y 305.583,Z 592.406,A -85,B 0,C 180,E1 -15853.296,E2 -15853.296} C_VEL
LIN {X 0,Y 305.587,Z 592.413,A -85,B 0,C 180,E1 -15856.021,E2 -15856.021} C_VEL
LIN {X 0,Y 305.571,Z 592.415,A -85,B 0,C 180,E1 -15859.446,E2 -15859.446} C_VEL
LIN {X 0,Y 305.484,Z 592.427,A -85,B 0,C 180,E1 -15863.042,E2 -15863.042} C_VEL
LIN {X 0,Y 305.542,Z 592.425,A -85,B 0,C 180,E1 -15866.228,E2 -15866.228} C_VEL
LIN {X 0,Y 305.491,Z 592.432,A -85,B 0,C 180,E1 -15869.051,E2 -15869.051} C_VEL
LIN {X 0,Y 305.44,Z 592.438,A -85,B 0,C 180,E1 -15871.953,E2 -15871.953} C_VEL
LIN {X 0,Y 305.458,Z 592.437,A -85,B 0,C 180,E1 -15875.114,E2 -15875.114} C_VEL
LIN {X 0,Y 305.489,Z 592.43,A -85,B 0,C 180,E1 -15878.54,E2 -15878.54} C_VEL
LIN {X 0,Y 305.504,Z 592.432,A -85,B 0,C 180,E1 -15882.597,E2 -15882.597} C_VEL
LIN {X 0,Y 305.484,Z 592.434,A -85,B 0,C 180,E1 -15886.357,E2 -15886.357} C_VEL
LIN {X 0,Y 305.464,Z 592.436,A -85,B 0,C 180,E1 -15889.895,E2 -15889.895} C_VEL
LIN {X 0,Y 305.512,Z 592.576,A -85,B 0,C 180,E1 -15891.318,E2 -15891.318} C_VEL
LIN {X 0,Y 308.322,Z 602.803,A -85,B 0,C 180,E1 -15894.863,E2 -15894.863} C_VEL
LIN {X 0,Y 310.551,Z 612.368,A -85,B 0,C 180,E1 -15897.872,E2 -15897.872} C_VEL
LIN {X 0,Y 312.368,Z 622.081,A -85,B 0,C 180,E1 -15900.683,E2 -15900.683} C_VEL
LIN {X 0,Y 312.3,Z 624.681,A -85,B 0,C 180,E1 -15901.361,E2 -15901.361} C_VEL
LIN {X 0,Y 311.707,Z 628.058,A -85,B 0,C 180,E1 -15902.183,E2 -15902.183} C_VEL
LIN {X 0,Y 315.608,Z 649.725,A -85,B 0,C 180,E1 -15903.316,E2 -15903.316} C_VEL
LIN {X 0,Y 317.679,Z 664.34,A -85,B 0,C 180,E1 -15903.981,E2 -15903.981} C_VEL
LIN {X 0,Y 319.554,Z 682.885,A -85,B 0,C 180,E1 -15904.726,E2 -15904.726} C_VEL
LIN {X 0,Y 317.548,Z 740.029,A -85,B 0,C 180,E1 -15906.22,E2 -15906.22} C_VEL
LIN {X 0,Y 316.404,Z 753.902,A -85,B 0,C 180,E1 -15906.824,E2 -15906.824} C_VEL
LIN {X 0,Y 314.956,Z 766.43,A -85,B 0,C 180,E1 -15907.621,E2 -15907.621} C_VEL
LIN {X 0,Y 313.352,Z 778.127,A -85,B 0,C 180,E1 -15908.626,E2 -15908.626} C_VEL
LIN {X 0,Y 311.566,Z 789.529,A -85,B 0,C 180,E1 -15909.88,E2 -15909.88} C_VEL
LIN {X 0,Y 309.813,Z 799.899,A -85,B 0,C 180,E1 -15911.312,E2 -15911.312} C_VEL
LIN {X 0,Y 308.119,Z 809.911,A -85,B 0,C 180,E1 -15913.049,E2 -15913.049} C_VEL
LIN {X 0,Y 306.595,Z 819.205,A -85,B 0,C 180,E1 -15915.056,E2 -15915.056} C_VEL
LIN {X 0,Y 305.379,Z 826.531,A -85,B 0,C 180,E1 -15917.034,E2 -15917.034} C_VEL
LIN {X 0,Y 304.454,Z 833.305,A -85,B 0,C 180,E1 -15919.358,E2 -15919.358} C_VEL
LIN {X 0,Y 304.085,Z 837.828,A -85,B 0,C 180,E1 -15921.36,E2 -15921.36} C_VEL
LIN {X 0,Y 303.95,Z 841.99,A -85,B 0,C 180,E1 -15923.858,E2 -15923.858} C_VEL
LIN {X 0,Y 303.948,Z 844.311,A -85,B 0,C 180,E1 -15926.022,E2 -15926.022} C_VEL
LIN {X 0,Y 304.122,Z 845.174,A -85,B 0,C 180,E1 -15927.351,E2 -15927.351} C_VEL
LIN {X 0,Y 304.222,Z 845.627,A -85,B 0,C 180,E1 -15928.676,E2 -15928.676} C_VEL
LIN {X 0,Y 304.301,Z 845.671,A -85,B 0,C 180,E1 -15930,E2 -15930} C_VEL
LIN {X 0,Y 304.254,Z 845.265,A -85,B 0,C 180,E1 -15931.324,E2 -15931.324} C_VEL
LIN {X 0,Y 304.201,Z 844.408,A -85,B 0,C 180,E1 -15932.648,E2 -15932.648} C_VEL
LIN {X 0,Y 303.956,Z 841.143,A -85,B 0,C 180,E1 -15936.153,E2 -15936.153} C_VEL
LIN {X 0,Y 304.05,Z 837.428,A -85,B 0,C 180,E1 -15938.641,E2 -15938.641} C_VEL
LIN {X 0,Y 304.458,Z 833.263,A -85,B 0,C 180,E1 -15940.642,E2 -15940.642} C_VEL
LIN {X 0,Y 305.416,Z 826.913,A -85,B 0,C 180,E1 -15942.965,E2 -15942.965} C_VEL
LIN {X 0,Y 306.6,Z 820.036,A -85,B 0,C 180,E1 -15944.944,E2 -15944.944} C_VEL
LIN {X 0,Y 307.831,Z 812.72,A -85,B 0,C 180,E1 -15946.656,E2 -15946.656} C_VEL
LIN {X 0,Y 309.346,Z 804.656,A -85,B 0,C 180,E1 -15948.202,E2 -15948.202} C_VEL
LIN {X 0,Y 311.279,Z 794.314,A -85,B 0,C 180,E1 -15949.795,E2 -15949.795} C_VEL
LIN {X 0,Y 313.24,Z 782.693,A -85,B 0,C 180,E1 -15951.209,E2 -15951.209} C_VEL
LIN {X 0,Y 314.986,Z 771.103,A -85,B 0,C 180,E1 -15952.29,E2 -15952.29} C_VEL
LIN {X 0,Y 316.642,Z 757.826,A -85,B 0,C 180,E1 -15953.201,E2 -15953.201} C_VEL
LIN {X 0,Y 317.762,Z 745.574,A -85,B 0,C 180,E1 -15953.785,E2 -15953.785} C_VEL
LIN {X 0,Y 318.387,Z 730.364,A -85,B 0,C 180,E1 -15954.224,E2 -15954.224} C_VEL
LIN {X 0,Y 319.686,Z 679.738,A -85,B 0,C 180,E1 -15955.381,E2 -15955.381} C_VEL
LIN {X 0,Y 316.628,Z 650.517,A -85,B 0,C 180,E1 -15956.442,E2 -15956.442} C_VEL
LIN {X 0,Y 312.269,Z 621.539,A -85,B 0,C 180,E1 -15957.671,E2 -15957.671} C_VEL
LIN {X 0,Y 311.435,Z 618.293,A -85,B 0,C 180,E1 -15957.906,E2 -15957.906} C_VEL
LIN {X 0,Y 308.157,Z 603.765,A -85,B 0,C 180,E1 -15961.255,E2 -15961.255} C_VEL
LIN {X 0,Y 305.462,Z 592.437,A -85,B 0,C 180,E1 -15964.028,E2 -15964.028} C_VEL
LIN {X 0,Y 305.496,Z 592.432,A -85,B 0,C 180,E1 -15966.735,E2 -15966.735} C_VEL
LIN {X 0,Y 305.462,Z 592.433,A -85,B 0,C 180,E1 -15970.601,E2 -15970.601} C_VEL
LIN {X 0,Y 305.484,Z 592.432,A -85,B 0,C 180,E1 -15973.643,E2 -15973.643} C_VEL
LIN {X 0,Y 305.505,Z 592.428,A -85,B 0,C 180,E1 -15977.403,E2 -15977.403} C_VEL
LIN {X 0,Y 305.516,Z 592.422,A -85,B 0,C 180,E1 -15981.603,E2 -15981.603} C_VEL
LIN {X 0,Y 305.458,Z 592.42,A -85,B 0,C 180,E1 -15984.886,E2 -15984.886} C_VEL
LIN {X 0,Y 305.451,Z 592.438,A -85,B 0,C 180,E1 -15988.353,E2 -15988.353} C_VEL
LIN {X 0,Y 305.515,Z 592.41,A -85,B 0,C 180,E1 -15991.113,E2 -15991.113} C_VEL
LIN {X 0,Y 305.566,Z 592.423,A -85,B 0,C 180,E1 -15994.087,E2 -15994.087} C_VEL
LIN {X 0,Y 305.494,Z 592.415,A -85,B 0,C 180,E1 -15998.402,E2 -15998.402} C_VEL
LIN {X 0,Y 305.583,Z 592.418,A -85,B 0,C 180,E1 -16001.217,E2 -16001.217} C_VEL
LIN {X 0,Y 305.642,Z 592.401,A -85,B 0,C 180,E1 -16005.349,E2 -16005.349} C_VEL
LIN {X 0,Y 305.628,Z 592.405,A -85,B 0,C 180,E1 -16009.399,E2 -16009.399} C_VEL
LIN {X 0,Y 305.79,Z 592.375,A -85,B 0,C 180,E1 -16012.074,E2 -16012.074} C_VEL
LIN {X 0,Y 305.684,Z 592.41,A -85,B 0,C 180,E1 -16014.723,E2 -16014.723} C_VEL
LIN {X 0,Y 305.952,Z 592.352,A -85,B 0,C 180,E1 -16018.684,E2 -16018.684} C_VEL
LIN {X 0,Y 305.953,Z 592.373,A -85,B 0,C 180,E1 -16021.316,E2 -16021.316} C_VEL
LIN {X 0,Y 305.681,Z 592.384,A -85,B 0,C 180,E1 -16025.277,E2 -16025.277} C_VEL
LIN {X 0,Y 305.801,Z 592.388,A -85,B 0,C 180,E1 -16027.926,E2 -16027.926} C_VEL
LIN {X 0,Y 305.595,Z 592.401,A -85,B 0,C 180,E1 -16031.945,E2 -16031.945} C_VEL
LIN {X 0,Y 305.631,Z 592.413,A -85,B 0,C 180,E1 -16035.035,E2 -16035.035} C_VEL
LIN {X 0,Y 305.57,Z 592.407,A -85,B 0,C 180,E1 -16039.445,E2 -16039.445} C_VEL
LIN {X 0,Y 305.483,Z 592.427,A -85,B 0,C 180,E1 -16043.041,E2 -16043.041} C_VEL
LIN {X 0,Y 305.542,Z 592.421,A -85,B 0,C 180,E1 -16046.228,E2 -16046.228} C_VEL
LIN {X 0,Y 305.491,Z 592.422,A -85,B 0,C 180,E1 -16049.051,E2 -16049.051} C_VEL
LIN {X 0,Y 305.443,Z 592.437,A -85,B 0,C 180,E1 -16051.952,E2 -16051.952} C_VEL
LIN {X 0,Y 305.458,Z 592.428,A -85,B 0,C 180,E1 -16055.114,E2 -16055.114} C_VEL
LIN {X 0,Y 305.478,Z 592.433,A -85,B 0,C 180,E1 -16058.537,E2 -16058.537} C_VEL
LIN {X 0,Y 305.488,Z 592.4,A -85,B 0,C 180,E1 -16062.594,E2 -16062.594} C_VEL
LIN {X 0,Y 305.441,Z 592.428,A -85,B 0,C 180,E1 -16066.349,E2 -16066.349} C_VEL
LIN {X 0,Y 305.45,Z 592.436,A -85,B 0,C 180,E1 -16069.691,E2 -16069.691} C_VEL
LIN {X 0,Y 306.644,Z 595.573,A -85,B 0,C 180,E1 -16069.936,E2 -16069.936} C_VEL
LIN {X 0,Y 308.285,Z 598.35,A -85,B 0,C 180,E1 -16070.208,E2 -16070.208} C_VEL
LIN {X 0,Y 316.79,Z 613.955,A -85,B 0,C 180,E1 -16071.587,E2 -16071.587} C_VEL
LIN {X 0,Y 321.696,Z 624.098,A -85,B 0,C 180,E1 -16072.368,E2 -16072.368} C_VEL
LIN {X 0,Y 319.968,Z 685.689,A -85,B 0,C 180,E1 -16073.756,E2 -16073.756} C_VEL
LIN {X 0,Y 319.499,Z 698.609,A -85,B 0,C 180,E1 -16074.209,E2 -16074.209} C_VEL
LIN {X 0,Y 318.685,Z 711.382,A -85,B 0,C 180,E1 -16074.921,E2 -16074.921} C_VEL
LIN {X 0,Y 317.494,Z 723.308,A -85,B 0,C 180,E1 -16075.828,E2 -16075.828} C_VEL
LIN {X 0,Y 316.053,Z 734.838,A -85,B 0,C 180,E1 -16076.99,E2 -16076.99} C_VEL
LIN {X 0,Y 314.521,Z 744.747,A -85,B 0,C 180,E1 -16078.248,E2 -16078.248} C_VEL
LIN {X 0,Y 312.95,Z 753.73,A -85,B 0,C 180,E1 -16079.65,E2 -16079.65} C_VEL
LIN {X 0,Y 311.331,Z 762.483,A -85,B 0,C 180,E1 -16081.335,E2 -16081.335} C_VEL
LIN {X 0,Y 309.572,Z 770.865,A -85,B 0,C 180,E1 -16083.362,E2 -16083.362} C_VEL
LIN {X 0,Y 308.283,Z 776.521,A -85,B 0,C 180,E1 -16085.056,E2 -16085.056} C_VEL
LIN {X 0,Y 307.047,Z 781.963,A -85,B 0,C 180,E1 -16087.101,E2 -16087.101} C_VEL
LIN {X 0,Y 306.073,Z 786.145,A -85,B 0,C 180,E1 -16089.151,E2 -16089.151} C_VEL
LIN {X 0,Y 305.317,Z 789.203,A -85,B 0,C 180,E1 -16091.201,E2 -16091.201} C_VEL
LIN {X 0,Y 304.882,Z 790.694,A -85,B 0,C 180,E1 -16092.563,E2 -16092.563} C_VEL
LIN {X 0,Y 304.587,Z 791.707,A -85,B 0,C 180,E1 -16093.926,E2 -16093.926} C_VEL
LIN {X 0,Y 304.321,Z 792.468,A -85,B 0,C 180,E1 -16095.919,E2 -16095.919} C_VEL
LIN {X 0,Y 304.159,Z 792.32,A -85,B 0,C 180,E1 -16097.998,E2 -16097.998} C_VEL
LIN {X 0,Y 304.233,Z 790.681,A -85,B 0,C 180,E1 -16100.694,E2 -16100.694} C_VEL
LIN {X 0,Y 304.542,Z 788.104,A -85,B 0,C 180,E1 -16102.897,E2 -16102.897} C_VEL
LIN {X 0,Y 304.808,Z 785.071,A -85,B 0,C 180,E1 -16104.708,E2 -16104.708} C_VEL
LIN {X 0,Y 305.328,Z 780.71,A -85,B 0,C 180,E1 -16106.701,E2 -16106.701} C_VEL
LIN {X 0,Y 306.121,Z 774.092,A -85,B 0,C 180,E1 -16109.013,E2 -16109.013} C_VEL
LIN {X 0,Y 307.019,Z 766.892,A -85,B 0,C 180,E1 -16110.984,E2 -16110.984} C_VEL
LIN {X 0,Y 308.036,Z 759.532,A -85,B 0,C 180,E1 -16112.615,E2 -16112.615} C_VEL
LIN {X 0,Y 309.172,Z 750.643,A -85,B 0,C 180,E1 -16114.237,E2 -16114.237} C_VEL
LIN {X 0,Y 310.227,Z 740.826,A -85,B 0,C 180,E1 -16115.688,E2 -16115.688} C_VEL
LIN {X 0,Y 311.435,Z 729.52,A -85,B 0,C 180,E1 -16117.016,E2 -16117.016} C_VEL
LIN {X 0,Y 312.478,Z 717.868,A -85,B 0,C 180,E1 -16118.081,E2 -16118.081} C_VEL
LIN {X 0,Y 313.22,Z 704.983,A -85,B 0,C 180,E1 -16118.955,E2 -16118.955} C_VEL
LIN {X 0,Y 313.757,Z 691.588,A -85,B 0,C 180,E1 -16119.575,E2 -16119.575} C_VEL
LIN {X 0,Y 314.281,Z 665.321,A -85,B 0,C 180,E1 -16120.224,E2 -16120.224} C_VEL
LIN {X 0,Y 315.351,Z 617.119,A -85,B 0,C 180,E1 -16121.305,E2 -16121.305} C_VEL
LIN {X 0,Y 307.188,Z 596.744,A -85,B 0,C 180,E1 -16122.358,E2 -16122.358} C_VEL
LIN {X 0,Y 305.615,Z 592.415,A -85,B 0,C 180,E1 -16122.619,E2 -16122.619} C_VEL
LIN {X 0,Y 305.595,Z 592.416,A -85,B 0,C 180,E1 -16126.02,E2 -16126.02} C_VEL
LIN {X 0,Y 305.575,Z 592.421,A -85,B 0,C 180,E1 -16129.443,E2 -16129.443} C_VEL
LIN {X 0,Y 305.511,Z 592.425,A -85,B 0,C 180,E1 -16130.933,E2 -16130.933} C_VEL
LIN {X 0,Y 307.489,Z 597.682,A -85,B 0,C 180,E1 -16131.252,E2 -16131.252} C_VEL
LIN {X 0,Y 316.059,Z 618.744,A -85,B 0,C 180,E1 -16132.425,E2 -16132.425} C_VEL
LIN {X 0,Y 314.219,Z 689.025,A -85,B 0,C 180,E1 -16134.2,E2 -16134.2} C_VEL
LIN {X 0,Y 313.735,Z 702.309,A -85,B 0,C 180,E1 -16134.791,E2 -16134.791} C_VEL
LIN {X 0,Y 313.002,Z 713.643,A -85,B 0,C 180,E1 -16135.508,E2 -16135.508} C_VEL
LIN {X 0,Y 312.036,Z 725.763,A -85,B 0,C 180,E1 -16136.528,E2 -16136.528} C_VEL
LIN {X 0,Y 311.098,Z 735.797,A -85,B 0,C 180,E1 -16137.609,E2 -16137.609} C_VEL
LIN {X 0,Y 310.029,Z 740.718,A -85,B 0,C 180,E1 -16138.197,E2 -16138.197} C_VEL
LIN {X 0,Y 306.373,Z 748.405,A -85,B 0,C 180,E1 -16139.147,E2 -16139.147} C_VEL
LIN {X 0,Y 302.622,Z 755.624,A -85,B 0,C 180,E1 -16140.209,E2 -16140.209} C_VEL
LIN {X 0,Y 301.405,Z 759.749,A -85,B 0,C 180,E1 -16140.97,E2 -16140.97} C_VEL
LIN {X 0,Y 300.164,Z 768.685,A -85,B 0,C 180,E1 -16142.98,E2 -16142.98} C_VEL
LIN {X 0,Y 299.291,Z 774.943,A -85,B 0,C 180,E1 -16144.727,E2 -16144.727} C_VEL
LIN {X 0,Y 298.539,Z 781.001,A -85,B 0,C 180,E1 -16146.831,E2 -16146.831} C_VEL
LIN {X 0,Y 297.909,Z 785.616,A -85,B 0,C 180,E1 -16148.876,E2 -16148.876} C_VEL
LIN {X 0,Y 297.369,Z 789.828,A -85,B 0,C 180,E1 -16151.432,E2 -16151.432} C_VEL
LIN {X 0,Y 297.095,Z 791.916,A -85,B 0,C 180,E1 -16153.314,E2 -16153.314} C_VEL
LIN {X 0,Y 297.007,Z 793.223,A -85,B 0,C 180,E1 -16155.224,E2 -16155.224} C_VEL
LIN {X 0,Y 297.065,Z 793.739,A -85,B 0,C 180,E1 -16157.171,E2 -16157.171} C_VEL
LIN {X 0,Y 297.313,Z 793.405,A -85,B 0,C 180,E1 -16159.149,E2 -16159.149} C_VEL
LIN {X 0,Y 297.736,Z 792.161,A -85,B 0,C 180,E1 -16161.163,E2 -16161.163} C_VEL
LIN {X 0,Y 298.379,Z 789.956,A -85,B 0,C 180,E1 -16163.208,E2 -16163.208} C_VEL
LIN {X 0,Y 299.283,Z 785.924,A -85,B 0,C 180,E1 -16165.696,E2 -16165.696} C_VEL
LIN {X 0,Y 300.39,Z 781.024,A -85,B 0,C 180,E1 -16167.863,E2 -16167.863} C_VEL
LIN {X 0,Y 301.989,Z 774.097,A -85,B 0,C 180,E1 -16170.194,E2 -16170.194} C_VEL
LIN {X 0,Y 303.485,Z 766.859,A -85,B 0,C 180,E1 -16172.096,E2 -16172.096} C_VEL
LIN {X 0,Y 305.305,Z 757.452,A -85,B 0,C 180,E1 -16174.064,E2 -16174.064} C_VEL
LIN {X 0,Y 307.034,Z 747.863,A -85,B 0,C 180,E1 -16175.668,E2 -16175.668} C_VEL
LIN {X 0,Y 308.618,Z 737.445,A -85,B 0,C 180,E1 -16177.063,E2 -16177.063} C_VEL
LIN {X 0,Y 310.107,Z 725.712,A -85,B 0,C 180,E1 -16178.305,E2 -16178.305} C_VEL
LIN {X 0,Y 311.34,Z 713.912,A -85,B 0,C 180,E1 -16179.26,E2 -16179.26} C_VEL
LIN {X 0,Y 312.195,Z 700.925,A -85,B 0,C 180,E1 -16180.029,E2 -16180.029} C_VEL
LIN {X 0,Y 312.68,Z 689.16,A -85,B 0,C 180,E1 -16180.495,E2 -16180.495} C_VEL
LIN {X 0,Y 315.041,Z 625.278,A -85,B 0,C 180,E1 -16182.186,E2 -16182.186} C_VEL
LIN {X 0,Y 308.348,Z 611.328,A -85,B 0,C 180,E1 -16183.447,E2 -16183.447} C_VEL
LIN {X 0,Y 302.122,Z 600.276,A -85,B 0,C 180,E1 -16184.635,E2 -16184.635} C_VEL
LIN {X 0,Y 300.145,Z 596.877,A -85,B 0,C 180,E1 -16185.031,E2 -16185.031} C_VEL
LIN {X 0,Y 298.808,Z 594.346,A -85,B 0,C 180,E1 -16185.311,E2 -16185.311} C_VEL
LIN {X 0,Y 298.601,Z 593.292,A -85,B 0,C 180,E1 -16185.431,E2 -16185.431} C_VEL
LIN {X 0,Y 298.589,Z 593.293,A -85,B 0,C 180,E1 -16189.146,E2 -16189.146} C_VEL
LIN {X 0,Y 298.752,Z 593.272,A -85,B 0,C 180,E1 -16191.886,E2 -16191.886} C_VEL
LIN {X 0,Y 298.656,Z 593.281,A -85,B 0,C 180,E1 -16194.599,E2 -16194.599} C_VEL
LIN {X 0,Y 298.918,Z 593.251,A -85,B 0,C 180,E1 -16198.653,E2 -16198.653} C_VEL
LIN {X 0,Y 298.918,Z 593.249,A -85,B 0,C 180,E1 -16201.347,E2 -16201.347} C_VEL
LIN {X 0,Y 298.788,Z 593.258,A -85,B 0,C 180,E1 -16206.754,E2 -16206.754} C_VEL
LIN {X 0,Y 298.674,Z 593.273,A -85,B 0,C 180,E1 -16209.481,E2 -16209.481} C_VEL
LIN {X 0,Y 298.546,Z 593.282,A -85,B 0,C 180,E1 -16213.616,E2 -16213.616} C_VEL
LIN {X 0,Y 298.542,Z 593.286,A -85,B 0,C 180,E1 -16216.409,E2 -16216.409} C_VEL
LIN {X 0,Y 298.506,Z 593.295,A -85,B 0,C 180,E1 -16219.655,E2 -16219.655} C_VEL
LIN {X 0,Y 298.451,Z 593.3,A -85,B 0,C 180,E1 -16223.598,E2 -16223.598} C_VEL
LIN {X 0,Y 298.484,Z 593.3,A -85,B 0,C 180,E1 -16226.575,E2 -16226.575} C_VEL
LIN {X 0,Y 298.416,Z 593.313,A -85,B 0,C 180,E1 -16229.642,E2 -16229.642} C_VEL
LIN {X 0,Y 298.391,Z 593.314,A -85,B 0,C 180,E1 -16232.801,E2 -16232.801} C_VEL
LIN {X 0,Y 298.466,Z 593.303,A -85,B 0,C 180,E1 -16236.814,E2 -16236.814} C_VEL
LIN {X 0,Y 298.448,Z 593.306,A -85,B 0,C 180,E1 -16241.251,E2 -16241.251} C_VEL
LIN {X 0,Y 298.414,Z 593.316,A -85,B 0,C 180,E1 -16245.048,E2 -16245.048} C_VEL
LIN {X 0,Y 298.418,Z 593.316,A -85,B 0,C 180,E1 -16248.745,E2 -16248.745} C_VEL
LIN {X 0,Y 298.454,Z 593.448,A -85,B 0,C 180,E1 -16250.413,E2 -16250.413} C_VEL
LIN {X 0,Y 301.164,Z 603.024,A -85,B 0,C 180,E1 -16253.921,E2 -16253.921} C_VEL
LIN {X 0,Y 303.501,Z 612.938,A -85,B 0,C 180,E1 -16257.177,E2 -16257.177} C_VEL
LIN {X 0,Y 305.326,Z 622.096,A -85,B 0,C 180,E1 -16259.959,E2 -16259.959} C_VEL
LIN {X 0,Y 305.494,Z 626.293,A -85,B 0,C 180,E1 -16261.112,E2 -16261.112} C_VEL
LIN {X 0,Y 305.275,Z 627.359,A -85,B 0,C 180,E1 -16261.376,E2 -16261.376} C_VEL
LIN {X 0,Y 309.38,Z 649.574,A -85,B 0,C 180,E1 -16262.599,E2 -16262.599} C_VEL
LIN {X 0,Y 311.586,Z 665.448,A -85,B 0,C 180,E1 -16263.348,E2 -16263.348} C_VEL
LIN {X 0,Y 313.34,Z 684.419,A -85,B 0,C 180,E1 -16264.119,E2 -16264.119} C_VEL
LIN {X 0,Y 311.316,Z 738.943,A -85,B 0,C 180,E1 -16265.574,E2 -16265.574} C_VEL
